(* CODESYS project BasePpt.library
   Company: Vistaprint
   Version: 0.0.0.76
   Description: 0.0.0.76	- IBH simulation improvements
      0.0.0.75	- new BaseConcept and BaseElements
      	- add full simulation to IBH
      	- remove simulation from OVN
      	- JCL clears Cleaning request in OFFbusy and MaintenanceMode
      0.0.0.74	- new BaseConcept and BaseElements
      0.0.0.73	- new BaseConcept and BaseElements
      0.0.0.72	- new BaseElements
      0.0.0.71	- JCL fix, Oven tracking band2 must be off for 3 cycles
      0.0.0.70	- PBC: Different SheetToSheet times for Auto & Manual Mode
      	- JCL: Rework Manual behavior
      0.0.0.69	- JCL: Take the message buffer out of the CUR
      0.0.0.68	- JCL: Error Exit Error fixed
      0.0.0.67	- JCL: Fix for Manual Mode Exit
      0.0.0.66	- JCL: added EOFF, changed PON
      0.0.0.65	- Added new BaseElements
      	- better DeStacker error msg
      0.0.0.64	- Added new BaseElements
      	- Added Manual State to JCL
      	- Adapted UMC usage in all controllers
      0.0.0.63	- GRR only showing 1 error when connection lost
      0.0.0.62	- PBC: changed buffer counter to int
      0.0.0.61	- DeStacker checks if empty
      0.0.0.60	- when DoubleSheet only Warning when turned off on DeStacker
      0.0.0.59	- BCH can go back to RUN from ERROR
      0.0.0.58	- BCH + JCL fixes
      0.0.0.57	- option to not wait for paper in OVN.OFFBusy
      	- support AnalogValue on GRR
      0.0.0.56	- fixed OVN.OFFBusy time calculation
      0.0.0.55	- JCL check Jetter state in RUN
      	- latest BaseConcept and BaseElements
      	- OVN wait in OFFBusy until sheets are out
      0.0.0.54	- TCP - Fix for constant resend of command
      0.0.0.53	- fixes
      0.0.0.52	- TCP - Introduced automatic reconnect
      0.0.0.51	- PBC - Fix for StopDestacking and Manual mode.
      0.0.0.50	- OVN has TSTOP when settings change
      0.0.0.49	- Saber PBC StopBit modification, different PBC alarm handling
      0.0.0.48	- small fixes for DeStacker
      0.0.0.47	- GRR warning automatically disappear
      0.0.0.46	- TCP.CtrlInit-Added call to super
      0.0.0.45	- manual operation on GRR is only a WARNING
      0.0.0.44	- OVN recovers from EOFF by reconnecting IBHLink
      0.0.0.43	- ignore bolStopReleaseItems when in manual mode
      0.0.0.42	- namechange GRN to GRR, ToggleBit for GRR
      0.0.0.41   - StopReleaseItems for PBC
      0.0.0.40	- new BaseElements
      0.0.0.39	- added CtrlSIf and strFullName where missing, new libraries
      0.0.0.38	- Better GRN error msgs
      0.0.0.37	- PBC Fixes
      0.0.0.36	- PTS Error Message Fixed
      	- PBC EvaluateEject fix
      	- PST Eject paper if not finished
      0.0.0.35	- Add long term test to PTS
      0.0.0.34 	- Pts fix when using with Servo
      0.0.0.33 	- Upgraded to newest TC 3.1 4016.12
      	- Upgraded all Libraries
      0.0.0.32 - Bug fixes in PTS and POD
      0.0.0.31 - BaseElements V0.0.1.30 referred
      0.0.0.30 - updated Oven and IBH
      0.0.0.29 - Fix PTS warning bug
      0.0.0.28 - Added a new version of the PBC
      0.0.0.27 - added strFullName
      0.0.0.26 - Added RAX, POD, TCP, PST, Updated PBC, PTS
      0.0.0.25 - Added the newest Base + Elements + TC 3.1 4016.6
      0.0.0.24 - Added the newest Base + Elements
      0.0.0.23 - Updated to TwinCat 4016.5
      0.0.0.22 - FB_PTB Always SingleAnswer
      0.0.0.21 - Added newest Elemets Library 
      0.0.0.20 - Added newest Elemets Library and reworked CtrlInit
      0.0.0.19 - Added newest Elemets Library
      0.0.0.18 - Added newest revision of the PTS
      
      0.0.0.16 - Added new Base and Elements 
      0.0.0.15 - Added new Base and Elements 
      0.0.0.14 - Added new Base and Elements 
      0.0.0.13 - Added new Base and Elements 
      0.0.0.11 - Added new Base and Elements library
      0.0.0.10 - PCE: no EOFF State!! in EOFF go to OFF (in Always); Redo changes of 0.0.0.6; PTS.Always no EOFF; sta_OFFBusy in PTS reworked;
      0.0.0.9 - Merged the DeStacker MDC with the BasePpt MDC
      0.0.0.8 - Added newer Versions of libraries.
      0.0.0.7 - Added newer Versions of libraries.
      0.0.0.6 - Changes for Simualtion in MDC, sta_OFFBusy in PTB/MDC reworked; Always in PTB reworked;
      0.0.0.5 - Added new Base_PLC 0.3.4.1
      0.0.0.4 - Bug fixed in FB_PTB
      0.0.0.3 - Update to take the newest libraries 
      0.0.0.2 - Update to Base_PLC 0.3.3.2; Update to Base_Elements 0.0.0.9
   Author: pcipriano
   Title: BasePpt

Project tree, tasks and I/O mapping:
  libraries: Base_Elements, 0.0.1.50 (Vistaprint); Base_PLC, 0.3.5.12 (Vistaprint); Tc2_EtherCAT, 3.3.3.0 (Beckhoff Automation GmbH); Tc2_MC2, 3.3.8.0 (Beckhoff Automation GmbH); Tc2_S5S7Com, 3.3.0.0 (Beckhoff Automation GmbH); Tc2_Standard, 3.3.0.0 (Beckhoff Automation GmbH); Tc2_System, 3.3.8.1 (Beckhoff Automation GmbH); Tc2_TcpIp, 3.3.2.0 (Beckhoff Automation GmbH); Tc2_Utilities, 3.3.8.0 (Beckhoff Automation GmbH); Tc3_Interfaces, 3.3.0.0 (Beckhoff Automation GmbH); Tc3_MemMan, 3.3.1.0 (Beckhoff Automation GmbH); Tc3_Module, 3.3.6.0 (Beckhoff Automation GmbH)
  GVLs/
    global variables Constants
  POUs/
    Controller/
      Driver/
        IBH (IBH Link)/
          function block FB_IBH [ST]: Always, bitAccess, CtrlInit, CtrlSIf, FB_init, getCmdState, getCtrlSIf, setAckError, setAirflow, setBeltOn, setOff, setRun, setSpeed, setStandby, setTemp, sta_CONNECT, sta_CONNECTBusy, sta_DISCONNECT, sta_DISCONNECTBusy, sta_OFF, sta_OFFBusy, sta_PON, sta_PONBusy, sta_READ, sta_READBusy, sta_WRITE, sta_WRITEBusy, StateMachine
          global variables IBH_CmdState
          data type T_Ctrl_SIf_IBH
          data type T_Ctrl_SIf_IBH_Cfg
          data type T_Ctrl_SIf_IBH_Cur
          data type T_Ctrl_SIf_IBH_Par
        POD (PLCopen Driver)/
          data type E_AmpType
          data type E_POD_UseHomeSwitch
          data type E_ValueType
          function block FB_POD [ST]: AD_SIf, CtrlInit, CycleEndDuty, CycleStartDuty, getCmdState, sJobReadParameter, sJobReadParameterNC, sJobWriteParameter, sJobWriteParameterNC, sta_AbsMoveBusy, sta_Error, sta_HomeBusy, sta_ModMoveBusy, sta_NegJogBusy, sta_NegMoveBusy, sta_PosJogBusy, sta_PosMoveBusy, sta_PowerOff, sta_PowerOnBusy, sta_QStopBusy, sta_RelMoveBusy, sta_StopBusy, sta_WaitForJob, StateMachine, StateMachine_Service
          global variables POD_Cmd
          global variables POD_Const
          data type T_POD
          data type T_POD_Cfg
          data type T_POD_DigitalInputs
          data type T_POD_Error
          data type T_POD_Move
          data type T_POD_Service
          data type T_POD_StateMachine
          data type T_POD_Status
          data type T_POD_StatusWord
        PTR [Paper Tracker]/
          data type E_PTR_Status
          function block FB_PTR [ST]: BeltLength, EnterComplete, FB_init, Insert, PaperEntryOffset, PaperOnBelt, Pop, PositionList, Push, Reset, TimeBase
          data type T_PTR_STRUCT
        TCP (TCP communication driver)/
          data type E_ALM_TCP
          function block FB_TCP [ST]: Always, CtrlInit, CtrlSIf, CycleEndDuty, CycleStartDuty, FB_init, getCmdState, getCtrlSIf, M_Pop, M_Push, ReceiveDataSequence, SendDataSequence, sta_CLOSE, sta_CLOSEBusy, sta_CONNECT, sta_CONNECTBusy, sta_ERROR, sta_ERRORQuit, StateMachine
          data type ST_Header
          data type T_Ctrl_SIf_TCP
          data type T_Ctrl_SIf_TCP_Cfg
          data type T_Ctrl_SIf_TCP_Cur
          data type T_Ctrl_SIf_TCP_Par
          global variables TCP_CmdState
          global variables TCP_Constants
      Lvl0/
        GRR (Granulate Remote)/
          helper/
            function cycle_Grr [ST]
            function init_Grr [ST]
            data type T_GRR
            data type T_GRR_CTRL
            data type T_GRR_ID
            data type T_GRR_IO
          data type E_ALM_GRR
          function block FB_GRR [ST]: Always, CtrlSIf, FB_init, getCtrlSIf, IoInBridge, IoOutBridge, sta_ERROR, sta_ERRORQuit, sta_OFF, sta_OFFBusy, sta_PON, sta_PONBusy, sta_RUN, sta_RUNBusy, StateMachine
          data type T_Ctrl_SIf_GRR
          data type T_Ctrl_SIf_GRR_Cfg
          data type T_Ctrl_SIf_GRR_Cur
          data type T_Ctrl_SIf_GRR_In
          data type T_Ctrl_SIf_GRR_Out
          data type T_Ctrl_SIf_GRR_Par
        JCL (Jetter Client)/
          helper/
            function cycle_Jcl [ST]
            function init_Jcl [ST]
            data type T_JCL
            data type T_JCL_CTRL
            data type T_JCL_ID
            data type T_JCL_IO
          data type E_ALM_JCL
          function block FB_JCL [ST]: Always, checkChildAlmClass, cmdCALIBRATION, cmdCLEAN, cmdOFF, cmdPON, cmdRUN, cmdSTANDBY, CtrlInit, CtrlSIf, FB_init, getCmdState, getCtrlSIf, HandleReceiveData, RequestState, ResetAlarms, sta_CALIBRATION, sta_CALIBRATIONBusy, sta_CLEANING, sta_CLEANINGBusy, sta_CONNECTBusy, sta_EOFF, sta_EOFFBusy, sta_ERROR, sta_ERRORQuit, sta_MANUALMODE, sta_OFF, sta_OFFBusy, sta_PON, sta_PONBusy, sta_RUN, sta_RUNBusy, sta_STANDBY, sta_STANDBYBusy, StateMachine, TCP
          global variables JCL_CmdState
          global variables JCL_Constants
          data type T_Ctrl_SIf_JCL
          data type T_Ctrl_SIf_JCL_Cfg
          data type T_Ctrl_SIf_JCL_Cur
          data type T_Ctrl_SIf_JCL_Par
          data type T_JCL_AlmMsg
          data type T_JCL_Command
          data type T_JCL_PrintDone
          data type T_JCL_RequestCleaning
          data type T_JCL_State
          data type U_JCL_Message
        RAX(Rotative Axis)/
          data type E_ALM_RAX
          function block FB_RAX [ST]: Always, CtrlSIf, FB_init, getCmdState, getDirection, IoOutBridge, sta_EOFF, sta_EOFFBusy, sta_ERROR, sta_ERRORQuit, sta_INIT, sta_INITBusy, sta_JOG_NEG, sta_JOG_POS, sta_OFF, sta_OFFBusy, sta_POS, sta_POSBusy, sta_REL_POS, sta_REL_POSBusy, sta_STOP, sta_STOPBusy, sta_Turn, sta_TurnBusy, StateMachine
          function fSetPar [ST]
          global variables RAX_CmdState
          data type T_Ctrl_SIf_RAX
          data type T_Ctrl_SIf_RAX_Cfg
          data type T_Ctrl_SIf_RAX_Cur
          data type T_Ctrl_SIf_RAX_Ilk
          data type T_Ctrl_SIf_RAX_Par
      Lvl1/
        BCH (Barcode with DataChannel)/
          helper/
            function cycle_Bch [ST]
            function init_Bch [ST]
            data type T_BCH
            data type T_BCH_CTRL
            data type T_BCH_DATACHN
            data type T_BCH_ID
            data type T_BCH_IO
          global variables BCH_CmdState
          data type E_ALM_BCH
          function block FB_BCH [ST]: Always, BarcodeReader, CtrlInit, CtrlSIf, DataChannel, FB_init, getCmdState, getCtrlSIf, IoInBridge, sta_ERROR, sta_ERRORQuit, sta_OFF, sta_OFFBusy, sta_RUN, sta_RUNBusy, StateMachine
          data type T_Ctrl_SIf_BCH
          data type T_Ctrl_SIf_BCH_Cfg
          data type T_Ctrl_SIf_BCH_Cur
          data type T_Ctrl_SIf_BCH_In
          data type T_Ctrl_SIf_BCH_Par
        MDC [Malteser Drive Controller]/
          data type E_ALM_MDC
          function block FB_MDC [ST]: ActualPosition, Always, CtrlInit, CtrlSIf, Drive, FB_init, getCmdState, getCtrlSIf, GetTurningDirection, IncrementPosition, IoInBridge, IoOutBridge, SetPositionToGo, sta_ERROR, sta_ERRORQuit, sta_InitializeBusy, sta_InPosition, sta_InPositionBusy, sta_OFF, sta_OFFBusy, sta_PON, sta_PREPOSITION, sta_PREPOSITIONbusy, sta_StartTurnBusy, sta_TurnBusy, sta_TURNDONE, StateMachine
          global variables MDC_CmdState
          data type T_Ctrl_SIf_MDC
          data type T_Ctrl_SIf_MDC_Cfg
          data type T_Ctrl_SIf_MDC_Cur
          data type T_Ctrl_SIf_MDC_Ilk
          data type T_Ctrl_SIf_MDC_In
          data type T_Ctrl_SIf_MDC_Out
          data type T_Ctrl_SIf_MDC_Par
        OVN (Oven)/
          helper/
            function cycle_Ovn [ST]
            function init_Ovn [ST]
            data type T_OVN
            data type T_OVN_CTRL
            data type T_OVN_DATACHN
            data type T_OVN_ID
            data type T_OVN_IO
          data type E_ALM_OVN
          function block FB_MONITOR [ST]: resetTime
          function block FB_OVN [ST]: Always, checkParameter, chooseTesomaErrors, CtrlInit, CtrlSIf, DataChannel, FB_init, getCmdState, getCtrlSIf, IBH, sta_BELTONLY, sta_BELTONLYBusy, sta_ERROR, sta_ERRORQuit, sta_OFF, sta_OFFBusy, sta_PON, sta_PONBusy, sta_RUN, sta_RUNBusy, StateMachine
          function block FB_Tracker [ST]: addElement, DataChannel, deleteAll, deleteElement, distanceAfterOven_mm, distanceBeforeOven_mm, markAllTrash, moduleLength_mm, numberOfElements, numberOfModules, sampleTime_us, sendData, update
          global variables OVN_CmdState
          data type T_Ctrl_SIf_OVN
          data type T_Ctrl_SIf_OVN_Cfg
          data type T_Ctrl_SIf_OVN_Cur
          data type T_Ctrl_SIf_OVN_In
          data type T_Ctrl_SIf_OVN_Out
          data type T_Ctrl_SIf_OVN_Par
          data type T_Data
        PTA [Paper Transport Alignment]/
          helper/
            function cycle_Pta [ST]
            function init_Pta [ST]
            data type T_PTA
            data type T_PTA_CTRL
            data type T_PTA_ID
            data type T_PTA_IO
        PTB [Paper Transport Belt]/
          BeltParameterFunction/
            data type T_Belt_Cfg_Base
            data type T_Belt_Cur_Base
            data type T_Belt_Par_Base
          helper/
            function cycle_Ptb [ST]
            function init_Ptb [ST]
            data type T_PTB
            data type T_PTB_CTRL
            data type T_PTB_ID
            data type T_PTB_IO
          data type E_ALM_PTB
          data type E_BELT_DIRECTION
          data type E_PTB_MODE
          data type E_PTB_PaperDirection
          function block FB_PTB [ST]: Always, CalculateBeltParameter, CalculateModeParameter, CheckPumpState, cmd_OFF, cmd_RUN, cmd_STOP, CtrlInit, CtrlSIf, Drive, FB_init, getCmdState, getCtrlSIf, IoInBridge, IoOutBridge, PaperPositionHandling, PositionList, SetPumpComand, sta_EJECTPAPER, sta_EJECTPAPERbusy, sta_ERROR, sta_ERRORQuit, sta_OFF, sta_OFFBusy, sta_PON, sta_RUN, sta_RUNBusy, sta_STACKPAPER, sta_STACKPAPERbusy, sta_STOP, sta_STOPBusy, StateMachine, VacuumPump
          global variables PTB_CmdState
          data type T_Ctrl_SIf_PTB
          data type T_Ctrl_SIf_PTB_Cfg
          data type T_Ctrl_SIf_PTB_Cur
          data type T_Ctrl_SIf_PTB_Ilk
          data type T_Ctrl_SIf_PTB_In
          data type T_Ctrl_SIf_PTB_Out
          data type T_Ctrl_SIf_PTB_Par
      Lvl2/
        PBC [Paper Buffer Controller]/
          helper/
            function cycle_Pbc [ST]
            function init_Pbc [ST]
            data type T_PBC
            data type T_PBC_CTRL
            data type T_PBC_ID
            data type T_PBC_IO
          data type E_ALM_PBC
          function block FB_PBC [ST]: Always, Belt, CountPaper, CtrlInit, CtrlSIf, DeStacker, FB_init, getCmdState, getCtrlSIf, IoInBridge, IoOutBridge, PaperHight, PaperWidth, sta_ERROR, sta_ERRORQuit, sta_INITbusy, sta_OFF, sta_OFFBusy, sta_PON, sta_RUN, sta_RUNbusy, sta_STOP, sta_STOPbusy, StateMachine
          global variables PBC_CmdState
          data type T_Ctrl_SIf_PBC
          data type T_Ctrl_SIf_PBC_Cfg
          data type T_Ctrl_SIf_PBC_Cur
          data type T_Ctrl_SIf_PBC_Ilk
          data type T_Ctrl_SIf_PBC_In
          data type T_Ctrl_SIf_PBC_Out
          data type T_Ctrl_SIf_PBC_Par
        PCE [Paper Belt Corner Element]/
          helper/
            function cycle_Pce [ST]
            function init_Pce [ST]
            data type T_PCE
            data type T_PCE_CTRL
            data type T_PCE_ID
            data type T_PCE_IO
          data type E_ALM_PCE
          function block FB_PCE [ST]: Always, CtrlInit, CtrlSIf, DriveIn, DriveOut, FB_init, getCmdState, getCtrlSIf, IoInBridge, IoOutBridge, PaperExitValveActive, PaperInputValveActive, sta_ERROR, sta_ERRORQuit, sta_OFF, sta_OFFBusy, sta_PON, sta_RUN, sta_RUNBusy, sta_STOP, sta_STOPBusy, StateMachine
          global variables PCE_CmdState
          data type T_Ctrl_SIf_PCE
          data type T_Ctrl_SIf_PCE_Cfg
          data type T_Ctrl_SIf_PCE_Cur
          data type T_Ctrl_SIf_PCE_Ilk
          data type T_Ctrl_SIf_PCE_In
          data type T_Ctrl_SIf_PCE_Out
          data type T_Ctrl_SIf_PCE_Par
        PST [Paper Stacker]/
          helper/
            function cycle_Pst [ST]
            function init_Pst [ST]
            data type T_PST
            data type T_PST_CTRL
            data type T_PST_ID
            data type T_PST_IO
          data type E_ALM_PST
          function block FB_PST [ST]: Always, Belt, CtrlInit, CtrlSIf, FB_init, getCmdState, getCtrlSIf, IoInBridge, PaperStackSendFifo, sta_EJECTBusy, sta_OFF, sta_OFFBusy, sta_RUN, sta_RUNBusy, StateMachine
          global variables PST_CmdState
          data type T_Ctrl_SIf_PST
          data type T_Ctrl_SIf_PST_Cfg
          data type T_Ctrl_SIf_PST_Cur
          data type T_Ctrl_SIf_PST_In
          data type T_Ctrl_SIf_PST_Par
          data type T_ItemPaperInfo
        PTS [Paper Turning Station]/
          helper/
            function cycle_Pts [ST]
            function init_Pts [ST]
            data type T_PTS
            data type T_PTS_CTRL
            data type T_PTS_ID
            data type T_PTS_IO
          data type E_ALM_PTS
          data type E_PTS_MODE
          function block FB_PTS [ST]: Always, Belt, CalculateOutputDelay, ChangeDistributionModeParameter, CtrlInit, CtrlSIf, FB_init, getCmdState, getCtrlSIf, GetItemBusy, IoInBridge, IoOutBridge, Malteser, Servo, sta_ERROR, sta_ERRORQuit, sta_GetItemBusy, sta_InitializeBusy, sta_OFF, sta_OFFBusy, sta_PaperDelayBusy, sta_PON, sta_RUN, sta_RUNBusy, sta_STANDBY, sta_STANDBYBusy, sta_STOP, sta_STOPbusy, sta_TurnEmptyBusy, sta_TurnPaperBusy, sta_WaitPaper, sta_WaitPaperGone, StateMachine
          global variables PTS_CmdState
          global variables PTS_Persistent
          data type T_Ctrl_SIf_PTS
          data type T_Ctrl_SIf_PTS_Cfg
          data type T_Ctrl_SIf_PTS_Cur
          data type T_Ctrl_SIf_PTS_Ilk
          data type T_Ctrl_SIf_PTS_In
          data type T_Ctrl_SIf_PTS_Out
          data type T_Ctrl_SIf_PTS_Par
          data type T_PTS_InOutPositions
      Lvl3/
      Lvl4/
      Top/
      Utility/
        Data Channel/
          OvenMessage/
            function block FB_OvenSendDch [ST]: InitChannel, SendData
            global variables OvenConst
            data type T_Oven_DCH
            data type T_OvenSendData
        FiFo/
          function block FB_DataSetFifo [ST]: A_Add, A_Get, A_Remove, A_Reset
        LookupTable/
          function block FB_LookupTable [ST]: A_Add, A_LookupByKey, A_LookupByValue, A_RemoveKey, A_Reset
          global variables LUT_Constants
  Version/
    global variables Global_Version
*)

// POUs/Controller/Driver/IBH (IBH Link)/T_Ctrl_SIf_IBH
TYPE T_Ctrl_SIf_IBH :
STRUCT
	///configuration
	Cfg: T_Ctrl_SIf_IBH_Cfg;
	///parameter
	Par: T_Ctrl_SIf_IBH_Par;
	///current values
	Cur: T_Ctrl_SIf_IBH_Cur;
END_STRUCT
END_TYPE

// POUs/Controller/Driver/IBH (IBH Link)/T_Ctrl_SIf_IBH_Cfg
TYPE T_Ctrl_SIf_IBH_Cfg :
STRUCT
	/// Number of Modules in use, <= 8 
	uiNumberOfModules: UINT;
	/// IPv4 network address 
	tIpAddress: T_IPv4Addr;
	/// Remote (server) port address 
	udiPortAdress: UDINT;
	/// MPI device address 
	nDeviceAddress: BYTE;
	/// Read/write from/to datablock number 
	nDatablockNumber: BYTE;
	/// Maximum time allowed for the execution of the command 
	tTimeout: TIME;
	/// Write byte/word offset/start address 
	nWriteStartAddress: WORD;
	/// Read byte/word offset/start address 
	nReadStartAddress: WORD;
	uiByteOffset_rd_iStatus: UINT;
	uiByteOffset_rd_bOff: UINT;
	uiBitOffset_rd_bOff: UINT;
	uiByteOffset_rd_bBeltOn: UINT;
	uiBitOffset_rd_bBeltOn: UINT;
	uiByteOffset_rd_bManual: UINT;
	uiBitOffset_rd_bManual: UINT;
	uiByteOffset_rd_bRun: UINT;
	uiBitOffset_rd_bRun: UINT;
	uiByteOffset_rd_bSetParam: UINT;
	uiBitOffset_rd_bSetParam: UINT;
	uiByteOffset_rd_bGetParam: UINT;
	uiBitOffset_rd_bGetParam: UINT;
	uiByteOffset_rd_bAckError: UINT;
	uiBitOffset_rd_bAckError: UINT;
	uiByteOffset_rd_adiTemp_mc: UINT;
	uiByteOffset_rd_adiAir_p: UINT;
	uiByteOffset_rd_diSpeed_mm_min: UINT;
	uiByteOffset_rd_iErrorLevel: UINT;
	uiByteOffset_rd_iErrorID: UINT;
	uiByteOffset_rd_iErrorValue: UINT;
	uiByteOffset_wr_iOff: UINT;
	uiByteOffset_wr_iBeltOn: UINT;
	uiByteOffset_wr_iManual: UINT;
	uiByteOffset_wr_iRun: UINT;
	uiByteOffset_wr_iSetParam: UINT;
	uiByteOffset_wr_iGetParam: UINT;
	uiByteOffset_wr_iAckError: UINT;
	uiByteOffset_wr_adiTemp_mc: UINT;
	uiByteOffset_wr_adiAir_p: UINT;
	uiByteOffset_wr_diSpeed_mm_min: UINT;
END_STRUCT
END_TYPE

// POUs/Controller/Driver/IBH (IBH Link)/T_Ctrl_SIf_IBH_Cur
TYPE T_Ctrl_SIf_IBH_Cur :
STRUCT
END_STRUCT
END_TYPE

// POUs/Controller/Driver/IBH (IBH Link)/T_Ctrl_SIf_IBH_Par
TYPE T_Ctrl_SIf_IBH_Par :
STRUCT
END_STRUCT
END_TYPE

// POUs/Controller/Driver/POD (PLCopen Driver)/E_AmpType
TYPE E_AmpType :
(
	BOTH_ROT_LIN := 0,
	ROTARY_AMP := 1,
	LINEAR_AMP := 2
) USINT;
END_TYPE

// POUs/Controller/Driver/POD (PLCopen Driver)/E_POD_UseHomeSwitch
TYPE E_POD_UseHomeSwitch :
(
	FUB_Input := 0,
	HomeSwitch,
	/// internal IO 2 Home switch 					0: Switched off, 1: Switched on
	SI0,
	/// internal IO 16 SI0:				0: Switched off (Open),1: Switched on (Close)
	SI1,
	/// internal IO 17 SI0:				0: Switched off (Open),1: Switched on (Close)
	SI2,
	/// internal IO 18 SI0:			0: Switched off (Open),1: Switched on (Close)
	SI3,
	/// internal IO 19 SI0:				0: Switched off (Open),1: Switched on (Close)
	SI4,
	/// internal IO 20 SI0:					0: Switched off (Open),1: Switched on (Close)
	SI5,
	/// internal IO 21 SI0:	 				0: Switched off (Open),1: Switched on (Close)
	/// internal IO 22 SI0:					0: Switched off (Open),1: Switched on (Close)
	SI6
) USINT;
END_TYPE

// POUs/Controller/Driver/POD (PLCopen Driver)/E_ValueType
TYPE E_ValueType :
(
	TYPE_NOT_SPECIFIED := 0,
	TYPE_SINT := 1,
	TYPE_INT := 2,
	TYPE_DINT := 3,
	TYPE_USINT := 4,
	TYPE_UINT := 5,
	TYPE_UDINT := 6,
	TYPE_STRING := 7
) USINT;
END_TYPE

// POUs/Controller/Driver/POD (PLCopen Driver)/T_POD
TYPE T_POD :
STRUCT
	strAxisName: STRING(31);
	strState: STRING;
	strCmd: STRING;
	intCmd: INT;
	intServiceCmd: INT;
	stStatus: T_POD_Status;
	stMove: T_POD_Move;
	stErr: T_POD_Error;
	stCfg: T_POD_Cfg;
	stService: T_POD_Service;
END_STRUCT
END_TYPE

// POUs/Controller/Driver/POD (PLCopen Driver)/T_POD_Cfg
TYPE T_POD_Cfg :
STRUCT
	bolSimulation: BOOL;
	///>0 Homeposition set if calibsignal active
	lreHomePosition: LREAL;
	/// Home Mode
	eHomingMode: MC_HomingMode;
	/// define home switch: 0 use FUB input, 
	eUseHomeSwitch: E_POD_UseHomeSwitch;
END_STRUCT
END_TYPE

// POUs/Controller/Driver/POD (PLCopen Driver)/T_POD_DigitalInputs
TYPE T_POD_DigitalInputs :
STRUCT
	///0 N-OT: 	Negative limit switch 	0: Switched off, 1: Switched on
	bol_N_OT: BOOL;
	///1 P-OT: 	Positive limit switch 	0: Switched off, 1: Switched on
	bol_P_OT: BOOL;
	///2 Home switch 					0: Switched off, 1: Switched on
	bol_HomeSwitch: BOOL;
	///16 SI0:	CN1-13pin 				0: Switched off (Open),1: Switched on (Close)
	bol_SI0: BOOL;
	///17 SI1:	CN1-7pin 				0: Switched off (Open),1: Switched on (Close)
	bol_SI1: BOOL;
	///18 SI2:	CN1-8pin 				0: Switched off (Open),1: Switched on (Close)
	bol_SI2: BOOL;
	///19 SI3:	CN1-9pin 				0: Switched off (Open),1: Switched on (Close)
	bol_SI3: BOOL;
	///20 SI4:	CN1-10pin 				0: Switched off (Open),1: Switched on (Close)
	bol_SI4: BOOL;
	///21 SI5:	CN1-11pin 				0: Switched off (Open),1: Switched on (Close)
	bol_SI5: BOOL;
	///22 SI6:	CN1-12pin 				0: Switched off (Open),1: Switched on (Close)
	bol_SI6: BOOL;
END_STRUCT
END_TYPE

// POUs/Controller/Driver/POD (PLCopen Driver)/T_POD_Error
TYPE T_POD_Error :
STRUCT
	/// Reset failure
	bolErrAck: BOOL;
	/// atleast one failure active
	bolErrorActive: BOOL;
	/// error in MC fub error
	bolMCError: BOOL;
	/// error in NC (motion controller)
	bolNCError: BOOL;
	/// error in drive (ELMO)
	bolDriveError: BOOL;
	/// error ID
	dwoErrorID: DWORD;
END_STRUCT
END_TYPE

// POUs/Controller/Driver/POD (PLCopen Driver)/T_POD_Move
TYPE T_POD_Move :
STRUCT
	///target position [Units] 
	lreSetPos: LREAL;
	/// Direction used for Modulo position
	eDirection: MC_Direction;
	///set speed [Units/s] 
	lreSetSpeed: LREAL;
	///set acc  [Units/s^2] 
	lreSetAcc: LREAL;
	///set dec  [Units/s^2] 
	lreSetDec: LREAL;
	///set dec  [Units/s^2] quickstop
	lreSetDecFast: LREAL;
	///lreSetDec : DINT; //set dec  [Units/s^2] 
	lreSetJerk: LREAL;
	/// speed override for all drive commands (0 ≤Override≤ 100.0)
	lreSpeedOverride: LREAL := 100.0;
	lreSWLimitNeg_mm: LREAL;
	lreSWLimitPos_mm: LREAL;
	/// Actual position [Units] 
	lreActPos: LREAL;
	/// Actual modulo position [Units] 
	lreActModPos: LREAL;
	/// act speed [Units/s] 
	lreActVel: LREAL;
	/// [Nm] actual torque The torque actual value corresponds to the instantaneous torque in the drive motor. The value is given in units of per thousand of rated torque.
	lreActTorque: LREAL;
END_STRUCT
END_TYPE

// POUs/Controller/Driver/POD (PLCopen Driver)/T_POD_Service
TYPE T_POD_Service :
STRUCT
	/// Index of the object that should be written to.
	worIndex: WORD;
	/// Sub-index of the object that should be written to.
	bytSubIndex: BYTE;
	/// Address (pointer) of the send buffer.
	dwo_pSrcBuf: DWORD;
	/// Number (in bytes) of data to be sent.
	udi_cbBufLen: UDINT;
	/// value type
	eValueType: E_ValueType;
	/// parameter number of read/write NC parameters
	eNC_ParNumber: MC_AxisParameter;
	/// write/read value if dwo_pSrcBuf = 0
	strValue: STRING;
END_STRUCT
END_TYPE

// POUs/Controller/Driver/POD (PLCopen Driver)/T_POD_StateMachine
TYPE T_POD_StateMachine :
STRUCT
	///actual state
	intState: INT;
	///state of last cycle
	intStateLastCycle: INT;
	///save history backup p.e. in ERROR state
	intStateHistory: INT;
	///set state for next cycle
	intStateNext: INT;
END_STRUCT
END_TYPE

// POUs/Controller/Driver/POD (PLCopen Driver)/T_POD_Status
TYPE T_POD_Status :
STRUCT
	/// Hardware enable:0 = Open 1 = Closed  
	bolEnable: BOOL;
	/// 1 = Network initialized  
	bolNetwOk: BOOL;
	/// 1 = Initialization done 
	bolInitOk: BOOL;
	bolReady: BOOL;
	/// 1 = Controller switched on  
	bolCtrlOn: BOOL;
	/// 1 = Homing done  
	bolHomeOk: BOOL;
	/// 1 = In position (target position reached)  
	bolInPos: BOOL;
	/// 1 = Axis moving  
	bolMoving: BOOL;
	/// 1 = negativ endswitch active -> no movement negative allowed
	bolNegHWSwitch: BOOL;
	/// 1 = positive endswitch active -> no movement positive allowed
	bolPosHWSwitch: BOOL;
	/// 1 = negativ endswitch active -> no movement negative allowed
	bolNegSWSwitch: BOOL;
	/// 1 = positive endswitch active -> no movement positive allowed
	bolPosSWSwitch: BOOL;
	/// drive digital inputs of elmo drive
	stDigIn: T_POD_DigitalInputs;
END_STRUCT
END_TYPE

// POUs/Controller/Driver/POD (PLCopen Driver)/T_POD_StatusWord
TYPE T_POD_StatusWord :
STRUCT
	/// 0	Ready TO Switch on =1
	bolReadyToSwitchOn: BOOL;
	///1	Switched on =1
	bolSwitchedOn: BOOL;
	///2	Operation enabeld =1
	bolOperationEnabled: BOOL;
	///3	Fault/Fault Reaction
	bolFault: BOOL;
	///4	MainPower on =1
	bolMainPowerOn: BOOL;
	///5	Quickstop inaktive =1
	bolQuickStopInactive: BOOL;
	///6	Switch on disabled =1
	bolSwitchOnDisabled: BOOL;
	///7	Warning is occurred =1
	bolWarning: BOOL;
	///8	not used always 0
	bolBit08: BOOL;
	///9	The Remote bit is always set by the Elmo servo drive
	bolRemote: BOOL;
	///10	Target Reached
	bolTargetReached: BOOL;
	///11	Internal Limit active =1
	bolInternLimit: BOOL;
END_STRUCT
END_TYPE

// POUs/Controller/Driver/PTR [Paper Tracker]/E_PTR_Status
TYPE E_PTR_Status :
(
	EnterBusy,
	OnBelt,
	ExitBusy,
	Gone,
	ERROR,
	MAX_E_PTR_Status
);
END_TYPE

// POUs/Controller/Driver/PTR [Paper Tracker]/T_PTR_STRUCT
TYPE T_PTR_STRUCT :
STRUCT
	// [us] Time of the paper on the belt
	udiTimeOnBelt_us				: UDINT;
	// [mm] Position of the paper on the belt
	lrePositionOnBelt_mm			: LREAL;
	// [mm] Position of the paper on the belt Adjusted to the possible maximum
	lrePositionOnBeltAdjusted_mm	: LREAL;
	// Paper Item Id
	udiItemId						: UDINT;
	// Error	
	eStatus							: E_PTR_Status;
END_STRUCT
END_TYPE

// POUs/Controller/Driver/TCP (TCP communication driver)/E_ALM_TCP
TYPE E_ALM_TCP :
(
	SocketConnectionLost := 1,
	AddToSendBufferFailed := 2,
	RemoveFromSendBufferFailed := 3,
	GetFromSendBufferFailed := 4,
	AddToReceiveBufferFailed := 5,
	RemoveFromReceiveBufferFailed := 6,
	GetFromReceiveBufferFailed := 7,
	NotSent := 8,
	NoAckReceived := 9,
	FubErrorClientConnection := 10,
	FubErrorSendData := 11,
	FubErrorReceiveData := 12,
	MAX_E_ALM_TCP
) UINT;
END_TYPE

// POUs/Controller/Driver/TCP (TCP communication driver)/ST_Header
{attribute 'pack_mode' := '1'}
TYPE ST_Header :
STRUCT
	uinMsgId: UINT;
	udiMsgSize: UDINT;
END_STRUCT
END_TYPE

// POUs/Controller/Driver/TCP (TCP communication driver)/T_Ctrl_SIf_TCP
TYPE T_Ctrl_SIf_TCP :
STRUCT
	/// configuration
	Cfg: T_Ctrl_SIf_TCP_Cfg;
	/// parameter
	Par: T_Ctrl_SIf_TCP_Par;
	/// current values
	Cur: T_Ctrl_SIf_TCP_Cur;
	/// alarm number used in this controller
	Alm: ARRAY[1..(E_ALM_TCP.MAX_E_ALM_TCP - 1)] OF T_Ctrl_Alm;
END_STRUCT
END_TYPE

// POUs/Controller/Driver/TCP (TCP communication driver)/T_Ctrl_SIf_TCP_Cfg
TYPE T_Ctrl_SIf_TCP_Cfg :
STRUCT
	/// depending on the protocol an ACK is used or not
	bUsingAck: BOOL;
	/// Enable Auto Reconnect
	bolAutoReconnectEnable: BOOL;
END_STRUCT
END_TYPE

// POUs/Controller/Driver/TCP (TCP communication driver)/T_Ctrl_SIf_TCP_Cur
TYPE T_Ctrl_SIf_TCP_Cur :
STRUCT
	bolFubErrorActive: BOOL;
END_STRUCT
END_TYPE

// POUs/Controller/Driver/TCP (TCP communication driver)/T_Ctrl_SIf_TCP_Par
TYPE T_Ctrl_SIf_TCP_Par :
STRUCT
	strIPAdr: STRING(15);
	udiPort: UDINT;
	tTOConnection: TIME;
	tTOReceive: TIME;
	tTOSend: TIME;
	iMaxWaitTimeAck: TIME;
	iMaxSendTry: USINT;
END_STRUCT
END_TYPE

// POUs/Controller/Lvl0/GRR (Granulate Remote)/helper/T_GRR
TYPE T_GRR :
STRUCT
	io:		T_GRR_IO;
	ctrl:	T_GRR_CTRL;
	id:		T_GRR_ID;
END_STRUCT
END_TYPE

// POUs/Controller/Lvl0/GRR (Granulate Remote)/helper/T_GRR_CTRL
TYPE T_GRR_CTRL :
STRUCT
	fbGrr: FB_GRR;
END_STRUCT
END_TYPE

// POUs/Controller/Lvl0/GRR (Granulate Remote)/helper/T_GRR_ID
TYPE T_GRR_ID :
STRUCT
	Grr: INT;
END_STRUCT
END_TYPE

// POUs/Controller/Lvl0/GRR (Granulate Remote)/helper/T_GRR_IO
TYPE T_GRR_IO :
STRUCT
	Out_intCommand: REFERENCE TO INT;
	Out_intConveyorBelt: REFERENCE TO INT;
	Out_intPowderVibrator: REFERENCE TO INT;
	Out_intConveyorVibrator: REFERENCE TO INT;
	Out_intAnalogValue: REFERENCE TO INT;
	Out_uinFilterClearingCycleTime_min: REFERENCE TO UINT;
	Out_bolToggleBitGrr: REFERENCE TO BOOL;
	In_bolSystemOk: REFERENCE TO BOOL;
	In_bolMainPressureError: REFERENCE TO BOOL;
	In_bolEoffOrFuseOk: REFERENCE TO BOOL;
	In_bolPowderLowWarning: REFERENCE TO BOOL;
	In_bolAutoMode: REFERENCE TO BOOL;
	In_intState: REFERENCE TO INT;
	In_bolToggleBitGrn: REFERENCE TO BOOL;
	In_intMainPressure: REFERENCE TO INT;
END_STRUCT
END_TYPE

// POUs/Controller/Lvl0/GRR (Granulate Remote)/E_ALM_GRR
TYPE E_ALM_GRR :
(
	NONE := 1,
	SystemError := 2,
	MainPressureError := 3,
	EoffOrFuseError := 4,
	LowPowderWarning := 5,
	ManualOperation := 6,
	LostConnection := 7,
	MAX_E_ALM_GRR
) UINT;
END_TYPE

// POUs/Controller/Lvl0/GRR (Granulate Remote)/T_Ctrl_SIf_GRR
TYPE T_Ctrl_SIf_GRR :
STRUCT
	/// configuration
	Cfg: T_Ctrl_SIf_GRR_Cfg;
	/// parameter
	Par: T_Ctrl_SIf_GRR_Par;
	/// current values
	Cur: T_Ctrl_SIf_GRR_Cur;
	///io input
	In: T_Ctrl_SIf_GRR_In;
	///io output
	Out: T_Ctrl_SIf_GRR_Out;
	/// alarm number used in this controller
	Alm: ARRAY[1..(E_ALM_GRR.MAX_E_ALM_GRR - 1)] OF T_Ctrl_Alm;
END_STRUCT
END_TYPE

// POUs/Controller/Lvl0/GRR (Granulate Remote)/T_Ctrl_SIf_GRR_Cfg
TYPE T_Ctrl_SIf_GRR_Cfg :
STRUCT
	rMaxFreq_Hz: REAL;
END_STRUCT
END_TYPE

// POUs/Controller/Lvl0/GRR (Granulate Remote)/T_Ctrl_SIf_GRR_Cur
TYPE T_Ctrl_SIf_GRR_Cur :
STRUCT
	intMainPressure: INT;
END_STRUCT
END_TYPE

// POUs/Controller/Lvl0/GRR (Granulate Remote)/T_Ctrl_SIf_GRR_In
TYPE T_Ctrl_SIf_GRR_In :
STRUCT
	bolSystemOk				: T_Ctrl_IoBool;
	bolMainPressureError	: T_Ctrl_IoBool;
	bolEoffOrFuseOk			: T_Ctrl_IoBool;
	bolPowderLowWarning		: T_Ctrl_IoBool;
	bolAutoMode				: T_Ctrl_IoBool;
	intState				: T_Ctrl_IoInt;
	bolToggleBitGrn			: T_Ctrl_IoBool;
	intMainPressure			: T_Ctrl_IoInt;
END_STRUCT
END_TYPE

// POUs/Controller/Lvl0/GRR (Granulate Remote)/T_Ctrl_SIf_GRR_Out
TYPE T_Ctrl_SIf_GRR_Out :
STRUCT
	intCommand						: BASE_PLC.T_Ctrl_IoInt;
	intConveyorBelt					: T_Ctrl_IoInt;
	intPowderVibrator				: T_Ctrl_IoInt;
	intConveyorVibrator				: T_Ctrl_IoInt;
	intAnalogValue					: T_Ctrl_IoInt;
	uinFilterClearingCycleTime_min	: T_Ctrl_IoUint;
	bolToggleBitGrr					: T_Ctrl_IoBool;
END_STRUCT
END_TYPE

// POUs/Controller/Lvl0/GRR (Granulate Remote)/T_Ctrl_SIf_GRR_Par
TYPE T_Ctrl_SIf_GRR_Par :
STRUCT
	rConveyorBelt_Hz: REAL;
	rPowderVibrator_Hz: REAL;
	rConveyorVibrator_Hz: REAL;
	rAnalogValue_p: REAL;
	uinFilterClearingCycleTime_min: UINT;
END_STRUCT
END_TYPE

// POUs/Controller/Lvl0/JCL (Jetter Client)/helper/T_JCL
TYPE T_JCL :
STRUCT
	io: T_JCL_IO;
	ctrl: T_JCL_CTRL;
	id: T_JCL_ID;
END_STRUCT
END_TYPE

// POUs/Controller/Lvl0/JCL (Jetter Client)/helper/T_JCL_CTRL
TYPE T_JCL_CTRL :
STRUCT
	fbJcl: FB_JCL;
	fbJcl_Tcp: FB_TCP;
END_STRUCT
END_TYPE

// POUs/Controller/Lvl0/JCL (Jetter Client)/helper/T_JCL_ID
TYPE T_JCL_ID :
STRUCT
	Jcl: INT;
	Jcl_Tcp: INT;
END_STRUCT
END_TYPE

// POUs/Controller/Lvl0/JCL (Jetter Client)/helper/T_JCL_IO
TYPE T_JCL_IO :
STRUCT
END_STRUCT
END_TYPE

// POUs/Controller/Lvl0/JCL (Jetter Client)/E_ALM_JCL
TYPE E_ALM_JCL :
(
	NONE := 1,
	JetterNotRun := 2,
	JetterManualWarning := 3,
	JetterManualError := 4,
	JetterEOff := 5,
	JetterCommunicationLost := 6,
	MAX_E_ALM_JCL
) UINT;
END_TYPE

// POUs/Controller/Lvl0/JCL (Jetter Client)/T_Ctrl_SIf_JCL
TYPE T_Ctrl_SIf_JCL :
STRUCT
	/// configuration
	Cfg: T_Ctrl_SIf_JCL_Cfg;
	/// parameter
	Par: T_Ctrl_SIf_JCL_Par;
	/// current values
	Cur: T_Ctrl_SIf_JCL_Cur;
	/// alarm number used in this controller
	Alm: ARRAY[1..(E_ALM_JCL.MAX_E_ALM_JCL - 1)] OF T_Ctrl_Alm;
END_STRUCT
END_TYPE

// POUs/Controller/Lvl0/JCL (Jetter Client)/T_Ctrl_SIf_JCL_Cfg
TYPE T_Ctrl_SIf_JCL_Cfg :
STRUCT
	/// FALSE = Do not allow manual mode, go to error if Jetter goes to manual / TRUE = Allow manual mode and stay in the last state 
	bolJetterManualModeAllowed: BOOL;
END_STRUCT
END_TYPE

// POUs/Controller/Lvl0/JCL (Jetter Client)/T_Ctrl_SIf_JCL_Cur
TYPE T_Ctrl_SIf_JCL_Cur :
STRUCT
	/// Additional states from TCP server
	/// Local control active. Commands from this client are ignored
	bolIsLocalControlled: BOOL;
	/// Remote control active. Commands from this client are accepted
	bolIsRemoteControlled: BOOL;
	/// Jetter ready for production
	bolReadyForProduction: BOOL;
	/// Print running, in production
	bolRunning: BOOL;
	/// System needs attention. Info or warning active
	bolNeedsAttention: BOOL;
	/// General error active
	bolError: BOOL;
	/// Cleaning cycle was aborted before finishing. Production not possible.
	bolCleaningIncomplete: BOOL;
	/// Print head needs cleaning.
	bolNeedsCleaning: BOOL;
	/// Timestamp of the last cleaning cycle. Format: YYYY-MM-DD-hh:mm:ss.xxx
	strDTOfLastCleaningCycle: STRING := '';
	/// Jetter state
	intJETState: INT;
END_STRUCT
END_TYPE

// POUs/Controller/Lvl0/JCL (Jetter Client)/T_Ctrl_SIf_JCL_Par
TYPE T_Ctrl_SIf_JCL_Par :
STRUCT
END_STRUCT
END_TYPE

// POUs/Controller/Lvl0/JCL (Jetter Client)/T_JCL_AlmMsg
TYPE T_JCL_AlmMsg :
STRUCT
	stHeader: ST_Header;
	/// Unique alarm number
	udiAlarmID: UDINT;
	/// Additional information
	udiInfo: UDINT;
	/// Corresponding alarm class
	usiClass: USINT;
	/// Corresponding controller ID
	uinCtrlID: UINT;
	/// Entry date and time
	strDTEntry: STRING(25);
	/// Alarm Text
	strText: STRING(255);
END_STRUCT
END_TYPE

// POUs/Controller/Lvl0/JCL (Jetter Client)/T_JCL_Command
{attribute 'pack_mode' := '1'}
TYPE T_JCL_Command :
STRUCT
	stHeader: ST_Header;
	usiCommand: USINT;
END_STRUCT
END_TYPE

// POUs/Controller/Lvl0/JCL (Jetter Client)/T_JCL_PrintDone
TYPE T_JCL_PrintDone :
STRUCT
	stHeader: ST_Header;
	usiBarcode: ARRAY[0..9] OF USINT;
	///  [%]
	usiInkLevelMainTank: USINT;
	///  [%]	
	usiInkLevelSupplyPrintModule1: USINT;
	///  [%]	
	usiInkLevelSupplyPrintModule2: USINT;
	///  [%]	
	usiInkLevelReturnPrintModule1: USINT;
	///  [%]	
	usiInkLevelReturnPrintModule2: USINT;
	///  [0.01 mbar]
	udiInkMeniscus: ARRAY[0..1] OF UDINT;
	///  [0.1 °C] 
	udiPrintHeadTemperature: ARRAY[0..1, 0..4] OF UDINT;
	///  [Micrometer]	//  Dimension of printed file calculated by DJM
	udiPrintWidthCalc: UDINT;
	///  [Micrometer]	//  Dimension of printed file calculated by DJM
	udiPrintLengthCalc: UDINT;
	///  [Micrometer]	//  Offset of print
	udiShiftXCalc: UDINT;
	///  [Micrometer]	//  Offset of print
	udiShiftYCalc: UDINT;
	///  [0.01°]		//  Offset of rotation angle 
	udiShiftAngleCalc: UDINT;
END_STRUCT
END_TYPE

// POUs/Controller/Lvl0/JCL (Jetter Client)/T_JCL_RequestCleaning
{attribute 'pack_mode' := '1'}
TYPE T_JCL_RequestCleaning :
STRUCT
	stHeader: ST_Header;
	/// Date and time of the last cleaning cycle
	strDTLastClean: STRING(25);
	/// Required interval for cleaning [min]
	uinRequiredInterval_min: UINT;
END_STRUCT
END_TYPE

// POUs/Controller/Lvl0/JCL (Jetter Client)/T_JCL_State
{attribute 'pack_mode' := '1'}
TYPE T_JCL_State :
STRUCT
	stHeader: ST_Header;
	usiMainState: USINT;
	///(Bit coded)	
	usiAddState: USINT;
END_STRUCT
END_TYPE

// POUs/Controller/Lvl0/JCL (Jetter Client)/U_JCL_Message
{attribute 'pack_mode' := '1'}
TYPE U_JCL_Message :

UNION
	Cmd: T_JCL_Command;
	State: T_JCL_State;
	PrintDone: T_JCL_PrintDone;
	ReqCleaning: T_JCL_RequestCleaning;
	AlmMsg: T_JCL_AlmMsg;
END_UNION

END_TYPE

// POUs/Controller/Lvl0/RAX(Rotative Axis)/E_ALM_RAX
{attribute 'qualified_only' := ''}
TYPE E_ALM_RAX :
(
	GeneralDrive := 1,
	GeneralNc,
	SwLimit,
	NegHwLimit,
	PosHwLimit,
	InterlockNegMove,
	InterlockPosMove,
	GeneralMCFUB,
	MAX_E_ALM
) UINT;
END_TYPE

// POUs/Controller/Lvl0/RAX(Rotative Axis)/T_Ctrl_SIf_RAX
TYPE T_Ctrl_SIf_RAX :
STRUCT
	///configuration
	Cfg: T_Ctrl_SIf_RAX_Cfg;
	///parameter
	Par: T_Ctrl_SIf_RAX_Par;
	///current values
	Cur: T_Ctrl_SIf_RAX_Cur;
	///alarm number used in this controller
	Alm: ARRAY[1..(E_ALM_RAX.MAX_E_ALM - 1)] OF T_Ctrl_Alm;
	///interlock of output/movements
	Ilk: T_Ctrl_SIf_RAX_Ilk;
END_STRUCT
END_TYPE

// POUs/Controller/Lvl0/RAX(Rotative Axis)/T_Ctrl_SIf_RAX_Cfg
TYPE T_Ctrl_SIf_RAX_Cfg :
STRUCT
	/// homing mode
	eHomingMode: MC_HomingMode;
	lreShortestWayWindow_deg: LREAL;
END_STRUCT
END_TYPE

// POUs/Controller/Lvl0/RAX(Rotative Axis)/T_Ctrl_SIf_RAX_Cur
TYPE T_Ctrl_SIf_RAX_Cur :
STRUCT
	/// [0.1°/s] current speed
	dinSpeed_0_1deg_s: DINT;
	/// [0.1°] current position
	dinPosition_0_1deg: DINT;
	/// [°] current modulo position
	dinModPosition_0_1deg: DINT;
	/// [0.1Nm] current torque
	dinTorque_0_1Nm: DINT;
	/// digital input1 from drive
	bol_di1: BOOL;
	/// digital input2 from drive
	bol_di2: BOOL;
	/// digital input3 from drive
	bol_di3: BOOL;
	/// digital input4 from drive
	bol_di4: BOOL;
	/// digital input5 from drive
	bol_di5: BOOL;
END_STRUCT
END_TYPE

// POUs/Controller/Lvl0/RAX(Rotative Axis)/T_Ctrl_SIf_RAX_Ilk
TYPE T_Ctrl_SIf_RAX_Ilk :
STRUCT
	/// interlock movment in positive direction
	bolMovePos: BOOL;
	/// interlock movment in negative direction
	bolMoveNeg: BOOL;
END_STRUCT
END_TYPE

// POUs/Controller/Lvl0/RAX(Rotative Axis)/T_Ctrl_SIf_RAX_Par
TYPE T_Ctrl_SIf_RAX_Par :
STRUCT
	/// [deg] home offset 
	dinHomeOffset_0_1deg: DINT;
	/// [0.1°] position init
	dinPositionInit_0_1deg: DINT;
	/// [0.1°] position absolute 
	dinPos_0_1deg: DINT;
	/// [0.1°] rel distance
	dinRelDist_0_1deg: DINT;
	/// [0.1°/s] position speed
	dinSpeed_0_1deg_s: DINT;
	///[%] percent from dinSetSpeed_0_1deg_s
	dinSpeed_per: DINT;
	/// [0.1°/s^2] position acceleration
	dintAccDec_0_1deg_s2: DINT;
	///[%] percent from dintAccDec_0_1deg_s2
	dinAcc_per: DINT;
	///[%] percent from dintAccDec_0_1deg_s2
	dinDec_per: DINT;
	/// [0.1°/s^2] position deceleration fast em stop
	dinSetDecFast_0_1deg_s2: DINT;
	/// [0.1°] negative sw limite
	dinSWLimitNeg_0_1deg: DINT;
	/// [0.1°] positive sw limite
	dinSWLimitPos_0_1deg: DINT;
END_STRUCT
END_TYPE

// POUs/Controller/Lvl1/BCH (Barcode with DataChannel)/helper/T_BCH
TYPE T_BCH :
STRUCT
	io: T_BCH_IO;
	ctrl: T_BCH_CTRL;
	id: T_BCH_ID;
	datachn: T_BCH_DATACHN;
END_STRUCT
END_TYPE

// POUs/Controller/Lvl1/BCH (Barcode with DataChannel)/helper/T_BCH_CTRL
TYPE T_BCH_CTRL :
STRUCT
	fbBch: FB_BCH;
	fbBch_Bcc: FB_BCC;
	fbBch_Bcc_Bcd: FB_BCD;
END_STRUCT
END_TYPE

// POUs/Controller/Lvl1/BCH (Barcode with DataChannel)/helper/T_BCH_DATACHN
TYPE T_BCH_DATACHN :
STRUCT
	rSendData: T_IdBaseSendData;
END_STRUCT
END_TYPE

// POUs/Controller/Lvl1/BCH (Barcode with DataChannel)/helper/T_BCH_ID
TYPE T_BCH_ID :
STRUCT
	Bch: INT;
	Bch_Bcc: INT;
	Bch_Bcc_Bcd: INT;
END_STRUCT
END_TYPE

// POUs/Controller/Lvl1/BCH (Barcode with DataChannel)/helper/T_BCH_IO
TYPE T_BCH_IO :
STRUCT
	In_bolSensorTrigScan: REFERENCE TO BOOL;
END_STRUCT
END_TYPE

// POUs/Controller/Lvl1/BCH (Barcode with DataChannel)/E_ALM_BCH
TYPE E_ALM_BCH :
(
	DataChannelMissing := 1,
	DataChannelBufferFull,
	BarcodeNotReadCorrectly,
	MAX_E_ALM_BCH
) UINT;
END_TYPE

// POUs/Controller/Lvl1/BCH (Barcode with DataChannel)/T_Ctrl_SIf_BCH
TYPE T_Ctrl_SIf_BCH :
STRUCT
	/// configuration
	Cfg: T_Ctrl_SIf_BCH_Cfg;
	/// parameter
	Par: T_Ctrl_SIf_BCH_Par;
	/// current values
	Cur: T_Ctrl_SIf_BCH_Cur;
	/// Input layer
	In: T_Ctrl_SIf_BCH_In;
	/// alarm number used in this controller
	Alm: ARRAY[1..(E_ALM_BCH.MAX_E_ALM_BCH - 1)] OF T_Ctrl_Alm;
END_STRUCT
END_TYPE

// POUs/Controller/Lvl1/BCH (Barcode with DataChannel)/T_Ctrl_SIf_BCH_Cfg
TYPE T_Ctrl_SIf_BCH_Cfg :
STRUCT
	/// TRUE = Enable Data Channel; False = Disable DataChannel
	bolEnableDataChannel			: BOOL;
	// TRUE = Negative Trigger Signal, FALSE = Positive Trigger Signal
	bolNegativeTriggerSignal 		: BOOL;
END_STRUCT
END_TYPE

// POUs/Controller/Lvl1/BCH (Barcode with DataChannel)/T_Ctrl_SIf_BCH_Cur
TYPE T_Ctrl_SIf_BCH_Cur :
STRUCT
END_STRUCT
END_TYPE

// POUs/Controller/Lvl1/BCH (Barcode with DataChannel)/T_Ctrl_SIf_BCH_In
TYPE T_Ctrl_SIf_BCH_In :
STRUCT
	/// Trigger the measurement sensor
	bolSensorTrigScan: BASE_PLC.T_Ctrl_IoBool;
END_STRUCT
END_TYPE

// POUs/Controller/Lvl1/BCH (Barcode with DataChannel)/T_Ctrl_SIf_BCH_Par
TYPE T_Ctrl_SIf_BCH_Par :
STRUCT
END_STRUCT
END_TYPE

// POUs/Controller/Lvl1/MDC [Malteser Drive Controller]/E_ALM_MDC
TYPE E_ALM_MDC :
(
	TableSensorTimeout 		:= 1,
	CrossSensorTimeout		:= 2,
	PositionSame			:= 3,
	MAX_E_ALM_MDC
);
END_TYPE

// POUs/Controller/Lvl1/MDC [Malteser Drive Controller]/T_Ctrl_SIf_MDC
TYPE T_Ctrl_SIf_MDC :
STRUCT
	///configuration
	Cfg: T_Ctrl_SIf_MDC_Cfg;
	///parameter
	Par: T_Ctrl_SIf_MDC_Par;
	///current values
	Cur: T_Ctrl_SIf_MDC_Cur;
	///io input
	In: T_Ctrl_SIf_MDC_In;
	///io output
	Out: T_Ctrl_SIf_MDC_Out;
	///alarm number used in this controller
	Alm: ARRAY[1..MAX_E_ALM_MDC] OF T_Ctrl_Alm;
	///interlock of output/movements
	Ilk: T_Ctrl_SIf_MDC_Ilk;
END_STRUCT
END_TYPE

// POUs/Controller/Lvl1/MDC [Malteser Drive Controller]/T_Ctrl_SIf_MDC_Cfg
TYPE T_Ctrl_SIf_MDC_Cfg :
STRUCT
	/// Number of positions in 360° of the Malteser drive
	uintPositionPerTurn		: UINT;
END_STRUCT
END_TYPE

// POUs/Controller/Lvl1/MDC [Malteser Drive Controller]/T_Ctrl_SIf_MDC_Cur
TYPE T_Ctrl_SIf_MDC_Cur :
STRUCT	
	/// Actual Position as position 
	uintActualPosition			: UINT;
	/// actual turning direction
	eActualTurningDirection		: E_TURN_DIRECTION;
	/// Reference still ok
	bolReferenceOk				: BOOL;		
END_STRUCT
END_TYPE

// POUs/Controller/Lvl1/MDC [Malteser Drive Controller]/T_Ctrl_SIf_MDC_Ilk
TYPE T_Ctrl_SIf_MDC_Ilk :
STRUCT
END_STRUCT
END_TYPE

// POUs/Controller/Lvl1/MDC [Malteser Drive Controller]/T_Ctrl_SIf_MDC_In
TYPE T_Ctrl_SIf_MDC_In :
STRUCT
	/// Is the cross in sensor positinon. One rotation step done.
	bolCrossPositionSensor				: BASE_PLC.T_Ctrl_IoBool;
	/// Is the table at 0° degrees
	bolTablePositionSensor				: BASE_PLC.T_Ctrl_IoBool;
END_STRUCT
END_TYPE

// POUs/Controller/Lvl1/MDC [Malteser Drive Controller]/T_Ctrl_SIf_MDC_Out
TYPE T_Ctrl_SIf_MDC_Out :
STRUCT
	intActualPosition		: BASE_PLC.T_Ctrl_IoInt;
END_STRUCT
END_TYPE

// POUs/Controller/Lvl1/MDC [Malteser Drive Controller]/T_Ctrl_SIf_MDC_Par
TYPE T_Ctrl_SIf_MDC_Par :
STRUCT
	/// <0 = Turn left; =0 automatic; >0 turn right
	intTurnDirection					: INT;
	/// Position to go to if comand turn is given. 0 = initialization position
	uinPositionToGo						: UINT;
	/// [ms] time to rotate one step 
	udiStepRotationTime_ms				: UDINT;
	/// [ms] initialization timeout time
	udiInitializationTime_ms			: UDINT;
	/// [ms] simulation time to rotate one step
	udiSimStepRotationTime_ms			: UDINT;
	/// [ms] simulation initialization timeout time
	udiSimInitializationTime_ms			: UDINT;
	/// [ms] simulation time to start rotate and Cross sensor needs to go away
	udiSimStartRotationTime_ms			: UDINT;
	/// [rpm] PrePosition Speed
	uinPrePositionSpeed_rpm				: UINT;
	/// [rpm] Position Speed
	uinPositionSpeed_rpm				: UINT;
END_STRUCT
END_TYPE

// POUs/Controller/Lvl1/OVN (Oven)/helper/T_OVN
TYPE T_OVN :
STRUCT
	io		: T_OVN_IO;
	ctrl	: T_OVN_CTRL;
	id		: T_OVN_ID;
	datachn	: T_OVN_DATACHN;
END_STRUCT
END_TYPE

// POUs/Controller/Lvl1/OVN (Oven)/helper/T_OVN_CTRL
TYPE T_OVN_CTRL :
STRUCT
	fbOvn: FB_OVN;
	fbOvn_Ibh: FB_IBH;
END_STRUCT
END_TYPE

// POUs/Controller/Lvl1/OVN (Oven)/helper/T_OVN_DATACHN
TYPE T_OVN_DATACHN :
STRUCT
	rSendData	: T_OvenSendData;
END_STRUCT
END_TYPE

// POUs/Controller/Lvl1/OVN (Oven)/helper/T_OVN_ID
TYPE T_OVN_ID :
STRUCT
	Ovn: INT;
	Ovn_Ibh: INT;
END_STRUCT
END_TYPE

// POUs/Controller/Lvl1/OVN (Oven)/helper/T_OVN_IO
TYPE T_OVN_IO :
STRUCT
	Out_uinBcrOvenAEvent: REFERENCE TO UINT;
	Out_udiBcrOvenACode: REFERENCE TO ULINT;
	Out_uinBcrOvenBEvent: REFERENCE TO UINT;
	Out_udiBcrOvenBCode: REFERENCE TO ULINT;
	In_bolBcrDistributionTrigger: REFERENCE TO BOOL;
	In_udiBarcode_new_1: REFERENCE TO ULINT;
	In_udiBarcode_new_2: REFERENCE TO ULINT;
	In_uinNew_element_1: REFERENCE TO UINT;
	In_uinNew_element_2: REFERENCE TO UINT;
	In_udiBarcode_delete_1: REFERENCE TO ULINT;
	In_udiBarcode_delete_2: REFERENCE TO ULINT;
	In_uinDelete_element_1: REFERENCE TO UINT;
	In_uinDelete_element_2: REFERENCE TO UINT;
END_STRUCT
END_TYPE

// POUs/Controller/Lvl1/OVN (Oven)/E_ALM_OVN
TYPE E_ALM_OVN :
(
	NONE := 0,
	TempError := 1,
	AirError := 2,
	SpeedError := 3,
	TimeoutError := 4,
	ParameterWarning := 5,
	ConnectionError := 6,
	WrongMode := 7,
	/// OvertemperaturePowerSection						- software reset	- operating mode must be reelected
	Tesoma10000 := 8,
	/// FailureOfActiveCoolingUnit
	Tesoma10002 := 9,
	/// ActiveCoolingUnitNotRunning
	Tesoma10003 := 10,
	/// FailureFuseGeneral													- transport starts immediately when sensor is free
	Tesoma10006 := 11,
	/// BeltPositionControlSensorError					- software reset
	Tesoma10010 := 12,
	/// BeltEdgeShutOff									- software reset
	Tesoma10011 := 13,
	/// FaultBeltSpeed									- software reset
	Tesoma10012 := 14,
	/// TransportOverload
	Tesoma10013 := 15,
	/// BeltControlDeviceFault							- software reset	- reset FC
	Tesoma10014 := 16,
	/// EmergencyStop														- would be resettable, but since power is gone, the acknowledge does not arrive
	Tesoma10016 := 17,
	/// BeltWearMonitor
	Tesoma10023 := 18,
	/// ControlCabinetFan
	Tesoma10024 := 19,
	/// ControlCabinetTemperatureTooHigh
	Tesoma10025 := 20,
	/// PowerSupplyFailure
	Tesoma10026 := 21,
	/// IntakeHoodTemperatureExceeded
	Tesoma10027 := 22,
	/// AirPressureTooLow
	Tesoma10030 := 23,
	/// BeltPositionControlNotWorking
	Tesoma10031 := 24,
	/// ErrorCoolingDeviceControlCabinet
	Tesoma10032 := 25,
	/// ControlCabinetCoolerAndSmallDrivesFuseFailure
	Tesoma10034 := 26,
	/// LimitSwitchingOff								- software reset	- after elimination, reactivates according zone
	Tesoma10x00 := 27,
	/// OvertemperatureStl								- software reset	- after elimination AND reset, the STL reactivates the accordant zone
	Tesoma10x01 := 28,
	/// FuseTriggered									- software reset	- after elimination, reactivates the accordant zone
	Tesoma10x02 := 29,
	/// FailureExhaustAirDps								- software reset	- after elimination, reactivates the accordant zone
	Tesoma10x03 := 30,
	/// ErrorFrequencyConverter							- software reset	- after elimination AND reset, the FC reactivates the accordant zone
	Tesoma10x07 := 31,
	/// TemperatureSensorIrDefective
	Tesoma10x13 := 32,
	/// FaultFrameCoolingSystemDps
	Tesoma10x14 := 33,
	/// FaultExhaustAirDps
	Tesoma10x15 := 34,
	/// TemperatureFault									- software reset
	Tesoma13x00 := 35,
	TesomaUnknown := 36,
	HostConnectionLost := 37,
	SettingsChanged := 38,
	MAX_E_ALM_OVN
);
END_TYPE

// POUs/Controller/Lvl1/OVN (Oven)/T_Ctrl_SIf_OVN
TYPE T_Ctrl_SIf_OVN :
STRUCT
	///configuration
	Cfg: T_Ctrl_SIf_OVN_Cfg;
	///parameter
	Par: T_Ctrl_SIf_OVN_Par;
	///current values
	Cur: T_Ctrl_SIf_OVN_Cur;
	///io input
	In: T_Ctrl_SIf_OVN_In;
	///io output
	Out: T_Ctrl_SIf_OVN_Out;
	///alarm number used in this controller
	Alm: ARRAY[1..(E_ALM_OVN.MAX_E_ALM_OVN - 1)] OF T_Ctrl_Alm;
END_STRUCT
END_TYPE

// POUs/Controller/Lvl1/OVN (Oven)/T_Ctrl_SIf_OVN_Cfg
TYPE T_Ctrl_SIf_OVN_Cfg EXTENDS T_Ctrl_SIf_MOD_Cfg :
STRUCT
	/// Number of Modules in use 
	uiNumberOfModules: UINT;
	/// Length of one Module 
	diModuleLength_mm: DINT;
	/// Distance before the first Module 
	diDistanceBeforeOven_mm: DINT;
	/// Distance after the last Module 
	diDistanceAfterOven_mm: DINT;
	/// Maximal Belt Speed in mm/min 
	diMaxSpeed_mm_min: DINT;
	/// Minimal Belt Speed in mm/min 
	diMinSpeed_mm_min: DINT;
	/// Minimal Temperature in deci °C 
	diMinTemp_dc: DINT;
	/// Maximal Temperature in deci °C 
	diMaxTemp_dc: DINT;
	/// Minimal Airflow in % 
	diMinAir_p: DINT;
	/// Maximal Airflow in % 
	diMaxAir_p: DINT;
	/// Auto Continue After Connection Error
	bAutoContinueAfterConnectionError: BOOL;
	/// Enable Data Channel
	bolDataChannelEnable: BOOL;
	/// ignore waiting for Paper to eject in OFFBusy
	bIgnoreOffBusyWaitPaper: BOOL;
END_STRUCT
END_TYPE

// POUs/Controller/Lvl1/OVN (Oven)/T_Ctrl_SIf_OVN_Cur
TYPE T_Ctrl_SIf_OVN_Cur EXTENDS T_Ctrl_SIf_MOD_Cur :
STRUCT
	/// Belt Speed in mm/min 
	diSpeed_mm_min: DINT;
	/// Temperature in deci °C 
	adiTemp_dc: ARRAY[0..(MAX_NUMBER_OF_OVEN_MODULES - 1)] OF DINT;
	/// Airflow in % 
	adiAir_p: ARRAY[0..(MAX_NUMBER_OF_OVEN_MODULES - 1)] OF DINT;
END_STRUCT
END_TYPE

// POUs/Controller/Lvl1/OVN (Oven)/T_Ctrl_SIf_OVN_In
TYPE T_Ctrl_SIf_OVN_In :
STRUCT
END_STRUCT
END_TYPE

// POUs/Controller/Lvl1/OVN (Oven)/T_Ctrl_SIf_OVN_Out
TYPE T_Ctrl_SIf_OVN_Out :
STRUCT
END_STRUCT
END_TYPE

// POUs/Controller/Lvl1/OVN (Oven)/T_Ctrl_SIf_OVN_Par
TYPE T_Ctrl_SIf_OVN_Par EXTENDS T_Ctrl_SIf_MOD_Par :
STRUCT
	/// Belt Speed in mm/min 
	diSpeed_mm_min: DINT;
	/// Belt Speed Band in mm/min 
	diSpeedBand1_mm_min: DINT;
	/// Belt Speed Band in mm/min 
	diSpeedBand2_mm_min: DINT;
	/// Belt Speed Timeout in ms 
	udiSpeedTimeout_ms: UDINT;
	/// Temperature in deci °C 
	adiTemp_dc: ARRAY[0..(MAX_NUMBER_OF_OVEN_MODULES - 1)] OF DINT;
	/// Temperature Band in deci °C 
	adiTempBand1_dc: ARRAY[0..(MAX_NUMBER_OF_OVEN_MODULES - 1)] OF DINT;
	/// Temperature Band in deci °C 
	adiTempBand2_dc: ARRAY[0..(MAX_NUMBER_OF_OVEN_MODULES - 1)] OF DINT;
	/// Temperature Timeout in ms 
	audiTempTimeout_ms: ARRAY[0..(MAX_NUMBER_OF_OVEN_MODULES - 1)] OF UDINT;
	/// Airflow in % 
	adiAir_p: ARRAY[0..(MAX_NUMBER_OF_OVEN_MODULES - 1)] OF DINT;
	/// Airflow Band in % 
	adiAirBand1_p: ARRAY[0..(MAX_NUMBER_OF_OVEN_MODULES - 1)] OF DINT;
	/// Airflow Band in % 
	adiAirBand2_p: ARRAY[0..(MAX_NUMBER_OF_OVEN_MODULES - 1)] OF DINT;
	/// Airflow Timeout in ms 
	audiAirTimeout_ms: ARRAY[0..(MAX_NUMBER_OF_OVEN_MODULES - 1)] OF UDINT;
	udiTimeoutOffBusy_ms: UDINT;
	udiTimeoutRunBusyReaction_ms: UDINT;
	udiTimeoutRunBusyInBand_ms: UDINT;
	udiTimeoutBeltOnlyReaction_ms: UDINT;
	udiTimeoutBeltOnlyBusy_ms: UDINT;
END_STRUCT
END_TYPE

// POUs/Controller/Lvl1/OVN (Oven)/T_Data
{attribute 'enable_dynamic_creation' := ''}
TYPE T_Data :
STRUCT
	uliBarcode: ULINT;
	bTrash: BOOL;
	diDistance_um: DINT;
	diSumTemp_mc: ARRAY[0..(MAX_NUMBER_OF_OVEN_MODULES - 1)] OF DINT;
	diCyclesInModule: ARRAY[0..(MAX_NUMBER_OF_OVEN_MODULES - 1)] OF DINT;
	bBarcodeMissed: BOOL;
END_STRUCT
END_TYPE

// POUs/Controller/Lvl1/PTA [Paper Transport Alignment]/helper/T_PTA
TYPE T_PTA :
STRUCT
	io:		T_PTA_IO;
	ctrl:	T_PTA_CTRL;
	id:		T_PTA_ID;
END_STRUCT
END_TYPE

// POUs/Controller/Lvl1/PTA [Paper Transport Alignment]/helper/T_PTA_CTRL
TYPE T_PTA_CTRL :
STRUCT
	fbPta: FB_PTB;	// PTA is a special type of PTB
	fbPta_Umc: FB_UMC;
END_STRUCT
END_TYPE

// POUs/Controller/Lvl1/PTA [Paper Transport Alignment]/helper/T_PTA_ID
TYPE T_PTA_ID :
STRUCT
	Pta: INT;
	Pta_Umc: INT;
END_STRUCT
END_TYPE

// POUs/Controller/Lvl1/PTA [Paper Transport Alignment]/helper/T_PTA_IO
TYPE T_PTA_IO :
STRUCT
	In_bolInputSensor: REFERENCE TO BOOL;
	In_bolOutputSensor: REFERENCE TO BOOL;
	
	In_uinUmc_Status: REFERENCE TO UINT;
	In_uinUmc_ActualSpeed: REFERENCE TO UINT;
	In_uinUmc_SetSpeed: REFERENCE TO UINT;
	In_uinUmc_IOData1: REFERENCE TO WORD;
	In_uinUmc_ECatState: REFERENCE TO UINT;
	In_strUmc_ECatNetId: REFERENCE TO AMSNETID;
	In_uinUmc_ECatPort: REFERENCE TO WORD;
	Out_uinUmc_Control: REFERENCE TO UINT;
	Out_uinUmc_SetSpeed: REFERENCE TO UINT;
END_STRUCT
END_TYPE

// POUs/Controller/Lvl1/PTB [Paper Transport Belt]/BeltParameterFunction/T_Belt_Cfg_Base
TYPE T_Belt_Cfg_Base :
STRUCT
	/// Assign the motor rotation to a belt direction.
	intForwardDirection				: INT;
	/// Assign the motor rotation to a belt direction.
	intBackwardDirection			: INT;
	/// [mm] the belt travels per motor rotation
	reaRpmDistance_mm					: REAL;
END_STRUCT
END_TYPE

// POUs/Controller/Lvl1/PTB [Paper Transport Belt]/BeltParameterFunction/T_Belt_Cur_Base
TYPE T_Belt_Cur_Base :
STRUCT
	/// [mm/s] Belt speed
	uinBeltSpeed_mms						: UINT;
	/// [rpm] Belt speed
	uinBeltSpeed_rpm						: UINT;
END_STRUCT
END_TYPE

// POUs/Controller/Lvl1/PTB [Paper Transport Belt]/BeltParameterFunction/T_Belt_Par_Base
TYPE T_Belt_Par_Base :
STRUCT
	/// eSpeedControlSelection.EFFECTIVE_SPEED : [mm/sec] Target speed. Uses reaRpmDistance_mm and uinLC11 to calculate the rpm
	uinBeltSpeed						: UINT;
	/// eSpeedControlSelection.EFFECTIVE_SPEED : [mm/sec] Target speed. Uses reaRpmDistance_mm and uinLC11 to calculate the rpm
	uinStackSpeed						: UINT;
END_STRUCT
END_TYPE

// POUs/Controller/Lvl1/PTB [Paper Transport Belt]/helper/T_PTB
TYPE T_PTB :
STRUCT
	io:		T_PTB_IO;
	ctrl:	T_PTB_CTRL;
	id:		T_PTB_ID;
END_STRUCT
END_TYPE

// POUs/Controller/Lvl1/PTB [Paper Transport Belt]/helper/T_PTB_CTRL
TYPE T_PTB_CTRL :
STRUCT
	fbPtb: FB_PTB;
	fbPtb_Umc: FB_UMC;
	fbPtb_Vpc: FB_VPC;
END_STRUCT
END_TYPE

// POUs/Controller/Lvl1/PTB [Paper Transport Belt]/helper/T_PTB_ID
TYPE T_PTB_ID :
STRUCT
	Ptb: INT;
	Ptb_Umc: INT;
	Ptb_Vpc: INT;
END_STRUCT
END_TYPE

// POUs/Controller/Lvl1/PTB [Paper Transport Belt]/helper/T_PTB_IO
TYPE T_PTB_IO :
STRUCT
	In_bolInputSensor: REFERENCE TO BOOL;
	In_bolOutputSensor: REFERENCE TO BOOL;
	
	In_bolVpc_VacuumSensor: REFERENCE TO BOOL;
	In_bolVpc_PumpOk: REFERENCE TO BOOL;
	Out_bolVpc_PumpOn: REFERENCE TO BOOL;	

	In_bolUmc_EmoOk: REFERENCE TO BOOL;
	In_uinUmc_Status: REFERENCE TO UINT;
	In_uinUmc_ActualSpeed: REFERENCE TO UINT;
	In_uinUmc_SetSpeed: REFERENCE TO UINT;
	In_uinUmc_IOData1: REFERENCE TO WORD;
	In_uinUmc_ECatState: REFERENCE TO UINT;
	In_strUmc_ECatNetId: REFERENCE TO AMSNETID;
	In_uinUmc_ECatPort: REFERENCE TO WORD;
	Out_uinUmc_Control: REFERENCE TO UINT;
	Out_uinUmc_SetSpeed: REFERENCE TO UINT;
END_STRUCT
END_TYPE

// POUs/Controller/Lvl1/PTB [Paper Transport Belt]/E_ALM_PTB
TYPE E_ALM_PTB :
(
	TestAlarm := 1,
	MAX_E_ALM_PTB 
);
END_TYPE

// POUs/Controller/Lvl1/PTB [Paper Transport Belt]/E_BELT_DIRECTION
TYPE E_BELT_DIRECTION :
(
	FORWARD			:= 0,
	BACKWARD		:= 1,
	MAX_E_BELT_DIRECTION
);
END_TYPE

// POUs/Controller/Lvl1/PTB [Paper Transport Belt]/E_PTB_MODE
TYPE E_PTB_MODE :
(
	Endless	,		// 0
	ToSensor,		// 1
	ToDistance,		// 2
	ToTime,			// 3
	Stack,			// 4
	MAX_E_PTB_MODE
);
END_TYPE

// POUs/Controller/Lvl1/PTB [Paper Transport Belt]/E_PTB_PaperDirection
TYPE E_PTB_PaperDirection :
(
	Portrait,
	Landscape,
	MAX_E_PTB_PaperDirection
);
END_TYPE

// POUs/Controller/Lvl1/PTB [Paper Transport Belt]/T_Ctrl_SIf_PTB
TYPE T_Ctrl_SIf_PTB :
STRUCT
	///configuration
	Cfg: T_Ctrl_SIf_PTB_Cfg;
	///parameter
	Par: T_Ctrl_SIf_PTB_Par;
	///current values
	Cur: T_Ctrl_SIf_PTB_Cur;
	///io input
	In: T_Ctrl_SIf_PTB_In;
	///io output
	Out: T_Ctrl_SIf_PTB_Out;
	///alarm number used in this controller
	Alm: ARRAY[1..E_ALM_PTB.MAX_E_ALM_PTB] OF T_Ctrl_Alm;
	///interlock of output/movements
	Ilk: T_Ctrl_SIf_PTB_Ilk;
END_STRUCT
END_TYPE

// POUs/Controller/Lvl1/PTB [Paper Transport Belt]/T_Ctrl_SIf_PTB_Cfg
TYPE T_Ctrl_SIf_PTB_Cfg :
STRUCT
	// Function Mode
	eMode							: E_PTB_MODE;
	// Vacuum pump present
	bolVacuumPresent				: BOOL;
	// [mm] Length of the belt
	udiBeltLength_mm				: UDINT;
	// Belt Parameter	
	rBeltParam						: T_Belt_Cfg_Base;
	// Enable Entry Belt Sensor Debounce
	bolEntrySensorDebounceEnable	: BOOL;
	// Enable Exit Belt Sensor Debounce
	bolExitSensorDebounceEnable		: BOOL;
END_STRUCT
END_TYPE

// POUs/Controller/Lvl1/PTB [Paper Transport Belt]/T_Ctrl_SIf_PTB_Cur
	TYPE T_Ctrl_SIf_PTB_Cur :
STRUCT	
	/// actual belt direction
	eActualDirection						: E_BELT_DIRECTION;
	/// [mm] Distance to move if Move Mode is distance
	udiDistanceToMove_mm					: UDINT;
	/// [ms] Time to move
	udiTimeToMove_ms						: UDINT;
	// Belt parameter
	rBeltParam								: T_Belt_Cur_Base;
	// Belt Run Time
	udiBeltTimeBase_mm						: UDINT;
	// Paper on the belt
	uinPaperOnBelt							: UINT;
	// Pointer to the Position list of the paper on the belt
	pPositionList							: POINTER TO T_PTR_STRUCT;
END_STRUCT
END_TYPE

// POUs/Controller/Lvl1/PTB [Paper Transport Belt]/T_Ctrl_SIf_PTB_Ilk
TYPE T_Ctrl_SIf_PTB_Ilk :
STRUCT
END_STRUCT
END_TYPE

// POUs/Controller/Lvl1/PTB [Paper Transport Belt]/T_Ctrl_SIf_PTB_In
TYPE T_Ctrl_SIf_PTB_In :
STRUCT
	bolBeltEntrySensor			: BASE_PLC.T_Ctrl_IoBool;
	bolBeltExitSensor			: BASE_PLC.T_Ctrl_IoBool;
	bolBeltEntrySensorPEdge		: BASE_PLC.T_Ctrl_IoBool;
	bolBeltEntrySensorNEdge		: BASE_PLC.T_Ctrl_IoBool;
	bolBeltExitSensorPEdge		: BASE_PLC.T_Ctrl_IoBool;
	bolBeltExitSensorNEdge		: BASE_PLC.T_Ctrl_IoBool;
END_STRUCT
END_TYPE

// POUs/Controller/Lvl1/PTB [Paper Transport Belt]/T_Ctrl_SIf_PTB_Out
TYPE T_Ctrl_SIf_PTB_Out :
STRUCT

END_STRUCT
END_TYPE

// POUs/Controller/Lvl1/PTB [Paper Transport Belt]/T_Ctrl_SIf_PTB_Par
TYPE T_Ctrl_SIf_PTB_Par :
STRUCT
	/// <0 = Backward; =0 None; >0 forward
	intDirection						: INT;
	/// [mm] Distance to move if Move Mode is distance
	udiDistanceToMove_mm				: UDINT;
	/// [ms] Time to move
	udiTimeToMove_ms					: UDINT;
	/// Stack hight in # of sheets
	uinPaperStackHight					: UINT;
	/// Automatic ejecting the paper if stackhight is reached
	bolAutoEjectAfterStack				: BOOL;
	/// Automatic stacking the paper after ejecting all paper
	bolAutoStackAfterEject				: BOOL;
	/// Belt Parameter
	rBeltParam							: T_Belt_Par_Base;
	// [ms] Stack delay time - Delay before out motor can move after paper entered system
	udiStackDelayTime_ms				: UDINT;
	// [mm] Belt Length
	udiBeltLength_mm					: UDINT;
	// Page running format
	ePaperOrientation					: E_PTB_PaperDirection;
	/// [mm] Paper Hight
	uinPaperHight_mm					: UINT;
	/// [mm] Paper Width
	uinPaperWidth_mm					: UINT;
	// [ms] Input Parameter Debounce time
	uinInputSignalDebounceTime_ms		: UINT;
END_STRUCT
END_TYPE

// POUs/Controller/Lvl2/PBC [Paper Buffer Controller]/helper/T_PBC
TYPE T_PBC :
STRUCT
	io: T_PBC_IO;
	ctrl: T_PBC_CTRL;
	id: T_PBC_ID;
END_STRUCT
END_TYPE

// POUs/Controller/Lvl2/PBC [Paper Buffer Controller]/helper/T_PBC_CTRL
TYPE T_PBC_CTRL :
STRUCT
	fbPbc_PtbDeStacker: FB_PTB;
	fbPbc_PtbDeStacker_Umc: FB_UMC;
	fbPbc_PtbBelt: FB_PTB;
	fbPbc_PtbBelt_Umc: FB_UMC;
	fbPbc_PtbBelt_Vpc: FB_VPC;
	fbPbc: FB_PBC;
END_STRUCT
END_TYPE

// POUs/Controller/Lvl2/PBC [Paper Buffer Controller]/helper/T_PBC_ID
TYPE T_PBC_ID :
STRUCT
	Pbc: INT;
	Pbc_PtbDeStacker: INT;
	Pbc_PtbDeStacker_Umc: INT;
	Pbc_PtbBelt: INT;
	Pbc_PtbBelt_Umc: INT;
	Pbc_PtbBelt_Vpc: INT;
END_STRUCT
END_TYPE

// POUs/Controller/Lvl2/PBC [Paper Buffer Controller]/helper/T_PBC_IO
TYPE T_PBC_IO :
STRUCT
	///TODO: describe why this is here
	In_bolPts_PaperSensor: REFERENCE TO BOOL;
	In_bolInputSensor: REFERENCE TO BOOL;
	In_bolOutputSensor: REFERENCE TO BOOL;
	In_bolCapacitySensor: REFERENCE TO BOOL;
	In_bolDoublePaperSensor: REFERENCE TO BOOL;
	In_bolAirPressureOk: REFERENCE TO BOOL;
	Out_bolAirPressureOn: REFERENCE TO BOOL;

	In_bolPtbBelt_Vpc_VacuumSensor: REFERENCE TO BOOL;
	In_bolPtbBelt_Vpc_PumpOk: REFERENCE TO BOOL;
	Out_bolPtbBelt_Vpc_PumpOn: REFERENCE TO BOOL;

	In_uinPtbBelt_Umc_Status: REFERENCE TO UINT;
	In_uinPtbBelt_Umc_ActualSpeed: REFERENCE TO UINT;
	In_uinPtbBelt_Umc_SetSpeed: REFERENCE TO UINT;
	In_uinPtbBelt_Umc_IOData1: REFERENCE TO WORD;
	In_uinPtbBelt_Umc_ECatState: REFERENCE TO UINT;
	In_strPtbBelt_Umc_ECatNetId: REFERENCE TO AMSNETID;
	In_uinPtbBelt_Umc_ECatPort: REFERENCE TO WORD;
	Out_uinPtbBelt_Umc_Control: REFERENCE TO UINT;
	Out_uinPtbBelt_Umc_SetSpeed: REFERENCE TO UINT;

	In_uinPtbDeStacker_Umc_Status: REFERENCE TO UINT;
	In_uinPtbDeStacker_Umc_ActualSpeed: REFERENCE TO UINT;
	In_uinPtbDeStacker_Umc_SetSpeed: REFERENCE TO UINT;
	In_uinPtbDeStacker_Umc_IOData1: REFERENCE TO WORD;
	In_uinPtbDeStacker_Umc_ECatState: REFERENCE TO UINT;
	In_strPtbDeStacker_Umc_ECatNetId: REFERENCE TO AMSNETID;
	In_uinPtbDeStacker_Umc_ECatPort: REFERENCE TO WORD;
	Out_uinPtbDeStacker_Umc_Control: REFERENCE TO UINT;
	Out_uinPtbDeStacker_Umc_SetSpeed: REFERENCE TO UINT;
END_STRUCT
END_TYPE

// POUs/Controller/Lvl2/PBC [Paper Buffer Controller]/E_ALM_PBC
TYPE E_ALM_PBC :
(
	PaperTransport := 1,
	BufferFull := 2,
	BufferEmpty := 3,
	DoublePaperError := 4,
	DataChannelBufferFull := 5,
	DataChannelSend := 6,
	PaperInject := 7,
	PaperInjectRetry := 8,
	DoNotReleaseItems := 9,
	DoublePaperWarning := 10,
	MAX_E_ALM_PBC
);
END_TYPE

// POUs/Controller/Lvl2/PBC [Paper Buffer Controller]/T_Ctrl_SIf_PBC
TYPE T_Ctrl_SIf_PBC :
STRUCT
	///configuration
	Cfg: T_Ctrl_SIf_PBC_Cfg;
	///parameter
	Par: T_Ctrl_SIf_PBC_Par;
	///current values
	Cur: T_Ctrl_SIf_PBC_Cur;
	///io input
	In: T_Ctrl_SIf_PBC_In;
	///io output
	Out: T_Ctrl_SIf_PBC_Out;
	///alarm number used in this controller
	Alm: ARRAY[1..E_ALM_PBC.MAX_E_ALM_PBC] OF T_Ctrl_Alm;
	///interlock of output/movements
	Ilk: T_Ctrl_SIf_PBC_Ilk;
END_STRUCT
END_TYPE

// POUs/Controller/Lvl2/PBC [Paper Buffer Controller]/T_Ctrl_SIf_PBC_Cfg
TYPE T_Ctrl_SIf_PBC_Cfg :
STRUCT
	/// True : Use the turn table sensor to detect ejects.
	bolUseTurnTableSensorForEject: BOOL;
	/// Enable the Data Channel to Saber to send the read barcodes to Saber
	bolEnableDataChannel: BOOL;
	/// Airpressure unit for the granulate available
	bolGranulatAirPressureUnitAvailable: BOOL;
	/// Enable or Disable the Saber Stop DeStack to do manual operation
	bolEnableSaberStopDeStack: BOOL;
END_STRUCT
END_TYPE

// POUs/Controller/Lvl2/PBC [Paper Buffer Controller]/T_Ctrl_SIf_PBC_Cur
TYPE T_Ctrl_SIf_PBC_Cur :
STRUCT
	/// How many papers are in the buffer. -1 = Paper count unknown
	intPaperInBufferCount: INT;
	/// Last Paper to eject count parameter
	uinPaperToEjectParameter: UINT;
	/// Actual count of the paper ejected 
	uinPaperToEjectCount: UINT;
	/// [ms] Time from sheet to sheet ejection in multi eject mode.
	uinSheetToSheetTime: UINT;
	/// Was paper before Eject available
	bolPaperBeforeEjectAvailable: BOOL;
	/// Paper to paper Timeout
	uinPaperToPaperTime_ms: UINT;
	/// Last Read Barcode			
	udiLastBarcode: UDINT;
	/// Total Paper Counter / Also used to signal a new Barcode read.			
	udiBarcodeChanged: UDINT;
END_STRUCT
END_TYPE

// POUs/Controller/Lvl2/PBC [Paper Buffer Controller]/T_Ctrl_SIf_PBC_Ilk
TYPE T_Ctrl_SIf_PBC_Ilk :
STRUCT
END_STRUCT
END_TYPE

// POUs/Controller/Lvl2/PBC [Paper Buffer Controller]/T_Ctrl_SIf_PBC_In
TYPE T_Ctrl_SIf_PBC_In :
STRUCT
	/// This sensor shows if the buffer reaches his capacity limits
	bolPaperAvailableExit: BASE_PLC.T_Ctrl_IoBool;
	/// Shows if there is paper available in the buffer
	bolPaperAvailableEntry: BASE_PLC.T_Ctrl_IoBool;
	/// Shows if there is a paper on the output of the buffer
	bolCapacityReached: BASE_PLC.T_Ctrl_IoBool;
	/// Double paper detection
	bolDoublePaperDetection: BASE_PLC.T_Ctrl_IoBool;
	/// Turn Table Mid Sensor
	bolTurnTableMiddleSensor: BASE_PLC.T_Ctrl_IoBool;
	/// Airpressure Ok
	bolAirPressorOk: BASE_PLC.T_Ctrl_IoBool;
END_STRUCT
END_TYPE

// POUs/Controller/Lvl2/PBC [Paper Buffer Controller]/T_Ctrl_SIf_PBC_Out
TYPE T_Ctrl_SIf_PBC_Out :
STRUCT
	/// Air on the Airpressure supply unit on:
	bolAirOn: BASE_PLC.T_Ctrl_IoBool;
END_STRUCT
END_TYPE

// POUs/Controller/Lvl2/PBC [Paper Buffer Controller]/T_Ctrl_SIf_PBC_Par
TYPE T_Ctrl_SIf_PBC_Par :
STRUCT
	/// [ms] Paper transport timeout - Time that paper is allowed to have for the transport to the front.
	udiPaperTransportTime: UDINT;
	/// Sheet to output with one run command.  0 = endless until stop
	udiSheetToEject: UDINT;
	/// [ms] Time from sheet to sheet ejection in multi eject mode in Auto Mode.
	udiSheetToSheetTime: UDINT;
	/// [ms] Time from sheet to sheet ejection in multi eject mode in Manual Mode.
	udiManualSheetToSheetTime_ms: UDINT;
	/// [ms] Paper transport time simulation
	udiSimPaperTransportTime: UDINT;
	/// [ms] Paper to paper transport time simulation
	udiSimPaperToPaperTransportTime: UDINT;
	/// # of retries for paper transport. 
	udiPaperInjectRetries: UDINT;
	/// Enable Double Paper detection
	bolEnableDoublePaperDetection: BOOL;
	/// [ms] Double Paper detection sensor debounce time
	udiDoublePaperDebounceTime_ms: UDINT;
	/// [ms] Retry Pause Time
	udiPaperInjectRetryPauseTime_ms: UDINT;
	/// Automatic or Manual DeStacking Mode
	bolAutomaticMode: BOOL;
	/// Indicates that the controller must not release any item but can still collect new items (RUN state). This flag is normally set by LineControl.
	bolStopReleaseItems: BOOL;
END_STRUCT
END_TYPE

// POUs/Controller/Lvl2/PCE [Paper Belt Corner Element]/helper/T_PCE
TYPE T_PCE :
STRUCT
	io:		T_PCE_IO;
	ctrl:	T_PCE_CTRL;
	id:		T_PCE_ID;
END_STRUCT
END_TYPE

// POUs/Controller/Lvl2/PCE [Paper Belt Corner Element]/helper/T_PCE_CTRL
TYPE T_PCE_CTRL :
STRUCT
	fbPce: FB_PCE;
	fbPce_PtbIn: FB_PTB;
	fbPce_PtbIn_Umc: FB_UMC;
	fbPce_PtbIn_Vpc: FB_VPC;
	fbPce_PtbOut: FB_PTB;
	fbPce_PtbOut_Umc: FB_UMC;
END_STRUCT
END_TYPE

// POUs/Controller/Lvl2/PCE [Paper Belt Corner Element]/helper/T_PCE_ID
TYPE T_PCE_ID :
STRUCT
	Pce: INT;
	Pce_PtbIn: INT;
	Pce_PtbIn_Umc: INT;
	Pce_PtbIn_Vpc: INT;
	Pce_PtbOut: INT;
	Pce_PtbOut_Umc: INT;
END_STRUCT
END_TYPE

// POUs/Controller/Lvl2/PCE [Paper Belt Corner Element]/helper/T_PCE_IO
TYPE T_PCE_IO :
STRUCT
	In_bolInputSensor: REFERENCE TO BOOL;
	In_bolOutputSensor: REFERENCE TO BOOL;
	In_bolCornerSensor: REFERENCE TO BOOL;
	Out_bolVacuumValveIn: REFERENCE TO BOOL;
	Out_bolVacuumValveOut: REFERENCE TO BOOL;

	In_uinUmcIn_Status: REFERENCE TO UINT;
	In_uinUmcIn_ActualSpeed: REFERENCE TO UINT;
	In_uinUmcIn_SetSpeed: REFERENCE TO UINT;
	In_uinUmcIn_IOData1: REFERENCE TO WORD;
	In_uinUmcIn_ECatState: REFERENCE TO UINT;
	In_strUmcIn_ECatNetId: REFERENCE TO AMSNETID;
	In_uinUmcIn_ECatPort: REFERENCE TO WORD;
	Out_uinUmcIn_Control: REFERENCE TO UINT;
	Out_uinUmcIn_SetSpeed: REFERENCE TO UINT;
	
	In_uinUmcOut_Status: REFERENCE TO UINT;
	In_uinUmcOut_ActualSpeed: REFERENCE TO UINT;
	In_uinUmcOut_SetSpeed: REFERENCE TO UINT;
	In_uinUmcOut_IOData1: REFERENCE TO WORD;
	In_uinUmcOut_ECatState: REFERENCE TO UINT;
	In_strUmcOut_ECatNetId: REFERENCE TO AMSNETID;
	In_uinUmcOut_ECatPort: REFERENCE TO WORD;
	Out_uinUmcOut_Control: REFERENCE TO UINT;
	Out_uinUmcOut_SetSpeed: REFERENCE TO UINT;
	
	In_bolVpc_VacuumSensor: REFERENCE TO BOOL;
	In_bolVpc_PumpOk: REFERENCE TO BOOL;
	Out_bolVpc_PumpOn: REFERENCE TO BOOL;
END_STRUCT
END_TYPE

// POUs/Controller/Lvl2/PCE [Paper Belt Corner Element]/E_ALM_PCE
TYPE E_ALM_PCE :
(
	PaperSensorError := 1,
	MAX_E_ALM_PCE
);
END_TYPE

// POUs/Controller/Lvl2/PCE [Paper Belt Corner Element]/T_Ctrl_SIf_PCE
TYPE T_Ctrl_SIf_PCE :
STRUCT
	///configuration
	Cfg: T_Ctrl_SIf_PCE_Cfg;
	///parameter
	Par: T_Ctrl_SIf_PCE_Par;
	///current values
	Cur: T_Ctrl_SIf_PCE_Cur;
	///io input
	In: T_Ctrl_SIf_PCE_In;
	///io output
	Out: T_Ctrl_SIf_PCE_Out;
	///alarm number used in this controller
	Alm: ARRAY[1..MAX_E_ALM_PCE] OF T_Ctrl_Alm;
	///interlock of output/movements
	Ilk: T_Ctrl_SIf_PCE_Ilk;
END_STRUCT
END_TYPE

// POUs/Controller/Lvl2/PCE [Paper Belt Corner Element]/T_Ctrl_SIf_PCE_Cfg
TYPE T_Ctrl_SIf_PCE_Cfg :
STRUCT
END_STRUCT
END_TYPE

// POUs/Controller/Lvl2/PCE [Paper Belt Corner Element]/T_Ctrl_SIf_PCE_Cur
TYPE T_Ctrl_SIf_PCE_Cur :
STRUCT
	/// [mm/s] Belt speed
	uinBeltSpeed: UINT;
END_STRUCT
END_TYPE

// POUs/Controller/Lvl2/PCE [Paper Belt Corner Element]/T_Ctrl_SIf_PCE_Ilk
TYPE T_Ctrl_SIf_PCE_Ilk :
STRUCT
END_STRUCT
END_TYPE

// POUs/Controller/Lvl2/PCE [Paper Belt Corner Element]/T_Ctrl_SIf_PCE_In
TYPE T_Ctrl_SIf_PCE_In :
STRUCT
	/// 0 = Paper not here; 1 = Paper detected
	bolPaperAvailable: BASE_PLC.T_Ctrl_IoBool;
END_STRUCT
END_TYPE

// POUs/Controller/Lvl2/PCE [Paper Belt Corner Element]/T_Ctrl_SIf_PCE_Out
TYPE T_Ctrl_SIf_PCE_Out :
STRUCT
	/// Paper Incoming Belt - 0 = Vacuum Valve Closed;  1 = Vacuum valve open
	bolVacuumValveIn: BASE_PLC.T_Ctrl_IoBool;
	/// Paper Outgoing Belt - 0 = Vacuum Valve Closed;  1 = Vacuum valve open
	bolVacuumValveOut: BASE_PLC.T_Ctrl_IoBool;
END_STRUCT
END_TYPE

// POUs/Controller/Lvl2/PCE [Paper Belt Corner Element]/T_Ctrl_SIf_PCE_Par
TYPE T_Ctrl_SIf_PCE_Par :
STRUCT
	/// [ms] Paper entry delay time. Time delay between detection and switching the vacuum
	uinPaperEntryDelayTime_ms: UDINT;
	/// [ms] Paper exit time
	uinPaperExitTime_ms: UDINT;
	/// [ms] Simulation Paper exit time
	uinSimPaperExitTime_ms: UDINT;
END_STRUCT
END_TYPE

// POUs/Controller/Lvl2/PST [Paper Stacker]/helper/T_PST
TYPE T_PST :
STRUCT
	io:		T_PST_IO;
	ctrl:	T_PST_CTRL;
	id:		T_PST_ID;
END_STRUCT
END_TYPE

// POUs/Controller/Lvl2/PST [Paper Stacker]/helper/T_PST_CTRL
TYPE T_PST_CTRL :
STRUCT
	fbPst: FB_PST;
	fbPst_Ptb: FB_PTB;
	fbPst_Ptb_Umc: FB_UMC;
	fbPst_Ptb_Vpc: FB_VPC;
END_STRUCT
END_TYPE

// POUs/Controller/Lvl2/PST [Paper Stacker]/helper/T_PST_ID
TYPE T_PST_ID :
STRUCT
	Pst: INT;
	Pst_Ptb: INT;
	Pst_Ptb_Umc: INT;
	Pst_Ptb_Vpc: INT;
END_STRUCT
END_TYPE

// POUs/Controller/Lvl2/PST [Paper Stacker]/helper/T_PST_IO
TYPE T_PST_IO :
STRUCT
	In_bolSensorPaperAtOperatorPos: REFERENCE TO BOOL;
	In_bolSensorStopperPosition: REFERENCE TO BOOL;
	In_bolSensorInfeed: REFERENCE TO BOOL;
	In_bolSensorOutfeed: REFERENCE TO BOOL;
	
	In_bolPtb_InputSensor: REFERENCE TO BOOL;
	In_bolPtb_OutputSensor: REFERENCE TO BOOL;
	
	In_bolPtb_Vpc_VacuumSensor: REFERENCE TO BOOL;
	In_bolPtb_Vpc_PumpOk: REFERENCE TO BOOL;
	Out_bolPtb_Vpc_PumpOn: REFERENCE TO BOOL;
	
	In_uinPtb_Umc_Status: REFERENCE TO UINT;
	In_uinPtb_Umc_ActualSpeed: REFERENCE TO UINT;
	In_uinPtb_Umc_SetSpeed: REFERENCE TO UINT;
	In_uinPtb_Umc_IOData1: REFERENCE TO WORD;
	In_uinPtb_Umc_ECatState: REFERENCE TO UINT;
	In_strPtb_Umc_ECatNetId: REFERENCE TO AMSNETID;
	In_uinPtb_Umc_ECatPort: REFERENCE TO WORD;
	Out_uinPtb_Umc_Control: REFERENCE TO UINT;
	Out_uinPtb_Umc_SetSpeed: REFERENCE TO UINT;
END_STRUCT
END_TYPE

// POUs/Controller/Lvl2/PST [Paper Stacker]/E_ALM_PST
TYPE E_ALM_PST :
(
	StackIncomplete := 1,
	NeedsEjectCommand := 2,
	StackOkButLastCodeNotRight := 3,
	StackNotOkButLastCodeRight := 4,
	ReadingBarcodeFailedAfterXRetries := 5,
	NewPaperDetectedDuringEjecting := 6,
	NewPaperDetectedWhileBarcodeReading := 7,
	MAX_E_ALM_PST
);
END_TYPE

// POUs/Controller/Lvl2/PST [Paper Stacker]/T_Ctrl_SIf_PST
TYPE T_Ctrl_SIf_PST :
STRUCT
	///configuration
	Cfg: T_Ctrl_SIf_PST_Cfg;
	///parameter
	Par: T_Ctrl_SIf_PST_Par;
	///current values
	Cur: T_Ctrl_SIf_PST_Cur;
	///io input
	In: T_Ctrl_SIf_PST_In;
	///alarm number used in this controller
	Alm: ARRAY[1..E_ALM_PST.MAX_E_ALM_PST] OF T_Ctrl_Alm;
END_STRUCT
END_TYPE

// POUs/Controller/Lvl2/PST [Paper Stacker]/T_Ctrl_SIf_PST_Cfg
TYPE T_Ctrl_SIf_PST_Cfg :
STRUCT
	/// Enable data channel to saber
	bolEnableDataChannel	: BOOL;
	/// Number of retry barcode read command if failed
	uinNumOfRetryRead		: UINT;
	/// Rotation direction for ejecting
	/// LEFT  = 1
	/// RIGHT = 2
	usiEjectingDirection	: INT;
	/// Rotation direction for reverse
	/// LEFT  = 1
	/// RIGHT = 2
	usiReverseDirection		: INT;
	/// Enable PST controlled Eject
	bolEnablePstEjectControl: BOOL;
END_STRUCT
END_TYPE

// POUs/Controller/Lvl2/PST [Paper Stacker]/T_Ctrl_SIf_PST_Cur
TYPE T_Ctrl_SIf_PST_Cur :
STRUCT
	/// # of papers in the stack
	uinStackHight: UINT;
	/// Total number of stacks ejected 
	udiNumOfStacksEjectedTotal: UDINT;
	/// Indicates that the last stacking job was incomplete. Run command not possible. Needs eject command from saber.
	bolStackIncomplete: BOOL;
END_STRUCT
END_TYPE

// POUs/Controller/Lvl2/PST [Paper Stacker]/T_Ctrl_SIf_PST_In
TYPE T_Ctrl_SIf_PST_In :
STRUCT
	/// Sensor detects if a paper is at the operator position
	bolSensorPaperAtOperatorPos: BASE_PLC.T_Ctrl_IoBoolDebounced;
	/// Sensor detects the stopper position (TRUE = stopper position down , FALSE = stopper position up)
	bolSensorStopperPosition: BASE_PLC.T_Ctrl_IoBoolDebounced;
	/// Sensor detects paper on outfeed position 
	bolSensorOutfeed: BASE_PLC.T_Ctrl_IoBoolDebounced;
	/// Sensor detects paper on infeed position
	bolSensorInfeed: BASE_PLC.T_Ctrl_IoBool;
END_STRUCT
END_TYPE

// POUs/Controller/Lvl2/PST [Paper Stacker]/T_Ctrl_SIf_PST_Par
TYPE T_Ctrl_SIf_PST_Par :
STRUCT
	/// Stack hight in # of paper to eject. Sent by saber. 
	uinStackHight: UINT;
	/// Last barcode in stack. Sent by saber. 
	/// If stack hight is reached and last barcode in stack detected, stacker automatically eject the whole stack.
	uliLastBarCodeInStack: ULINT;
	/// [mm/s] Belt reverse speed to bring stopper back to up position
	uinBeltReverseSpeed_mmsec: UINT;
	/// [mm/s] Belt speed for ejecting the whole stack
	uinBeltEjectSpeed_mmsec: UINT;
	/// [ms] Paper is at operator position delay time
	udiPaperAtOpPosDebounceTime_ms: UDINT;
	/// [ms] Stopper position delay time
	udiStopperPosDebounceTime_ms: UDINT;
	/// [ms] Outfeed sensor delay time
	udiSensorOutfeedDebounceTime_ms: UDINT;
	/// [ms] Stack eject delay time - Delay before belt starts to eject the stack if hight is reached.
	udiStackEjectDelayTime_ms: UDINT;
	/// [ms] Stack ejecting time - Time for how long the belt should move in eject direction 
	udiStackEjectingTime_ms: UDINT;
	/// [ms] Belt reverse delay time - Delay before belt starts moving backward after ejecting stack.
	udiBeltReverseDelayTime_ms: UDINT;
	/// [ms] Barcode reader trigger delay time - Delay time, until a read command will be executed, after a new paper was detected at infeed sensor.
	udiBarcodeReaderTriggerDelayTime_ms: UDINT;
	/// [ms] Simulation time paper infeed stroke
	udiSimTimePaperInfeedStroke_ms: UDINT;
END_STRUCT
END_TYPE

// POUs/Controller/Lvl2/PST [Paper Stacker]/T_ItemPaperInfo
{attribute 'enable_dynamic_creation' := ''}
TYPE T_ItemPaperInfo :
STRUCT
	/// Position in the stack
	uinPosInStack: UINT;
	/// Barcode of the paper
	uliBarCode: ULINT;
END_STRUCT
END_TYPE

// POUs/Controller/Lvl2/PTS [Paper Turning Station]/helper/T_PTS
TYPE T_PTS :
STRUCT
	io			: T_PTS_IO;
	ctrl		: T_PTS_CTRL;
	id			: T_PTS_ID;
END_STRUCT
END_TYPE

// POUs/Controller/Lvl2/PTS [Paper Turning Station]/helper/T_PTS_CTRL
TYPE T_PTS_CTRL :
STRUCT
	fbPts_RAX_POD		: FB_POD;
	fbPts_RAX			: FB_RAX;
	fbPts_Ptb			: FB_PTB;
	fbPts_Ptb_Umc		: FB_UMC;
	fbPts_Ptb_Vpc		: FB_VPC;
	fbPts_Mdc_Umc		: FB_UMC;
	fbPts_Mdc			: FB_MDC;
	fbPts				: FB_PTS;
END_STRUCT
END_TYPE

// POUs/Controller/Lvl2/PTS [Paper Turning Station]/helper/T_PTS_ID
TYPE T_PTS_ID :
STRUCT
	Pts				: INT;
	Pts_Ptb			: INT;
	Pts_Ptb_Umc		: INT;
	Pts_Ptb_Vpc		: INT;
	Pts_Mdc			: INT;
	Pts_Mdc_Umc		: INT;
	/// New Servo Drive PLC opend driver
	Pts_RAX_POD		: INT;
	/// New Servo Drive
	Pts_RAX			: INT;
END_STRUCT
END_TYPE

// POUs/Controller/Lvl2/PTS [Paper Turning Station]/helper/T_PTS_IO
TYPE T_PTS_IO :
STRUCT
	In_bolPaperSensor: REFERENCE TO BOOL;
	
	In_bolMdc_CrossPositionSensor: REFERENCE TO BOOL;
	In_bolMdc_TablePositionSensor: REFERENCE TO BOOL;
	
	In_uinMdc_Umc_Status: REFERENCE TO UINT;
	In_uinMdc_Umc_ActualSpeed: REFERENCE TO UINT;
	In_uinMdc_Umc_SetSpeed: REFERENCE TO UINT;
	In_uinMdc_Umc_IOData1: REFERENCE TO WORD;
	In_uinMdc_Umc_ECatState: REFERENCE TO UINT;
	In_strMdc_Umc_ECatNetId: REFERENCE TO AMSNETID;
	In_uinMdc_Umc_ECatPort: REFERENCE TO WORD;
	Out_uinMdc_Umc_Control: REFERENCE TO UINT;
	Out_uinMdc_Umc_SetSpeed: REFERENCE TO UINT;
	
	In_uinPtb_Umc_Status: REFERENCE TO UINT;
	In_uinPtb_Umc_ActualSpeed: REFERENCE TO UINT;
	In_uinPtb_Umc_SetSpeed: REFERENCE TO UINT;
	In_uinPtb_Umc_IOData1: REFERENCE TO WORD;
	In_uinPtb_Umc_ECatState: REFERENCE TO UINT;
	In_strPtb_Umc_ECatNetId: REFERENCE TO AMSNETID;
	In_uinPtb_Umc_ECatPort: REFERENCE TO WORD;
	Out_uinPtb_Umc_Control: REFERENCE TO UINT;
	Out_uinPtb_Umc_SetSpeed: REFERENCE TO UINT;
	
	In_bolPtb_Vpc_VacuumSensor: REFERENCE TO BOOL;
	In_bolPtb_Vpc_PumpOk: REFERENCE TO BOOL;
	Out_bolPtb_Vpc_PumpOn: REFERENCE TO BOOL;
	
	In_bolRax_PositionSensor: REFERENCE TO BOOL;
	//TODO
END_STRUCT
END_TYPE

// POUs/Controller/Lvl2/PTS [Paper Turning Station]/E_ALM_PTS
TYPE E_ALM_PTS :
(
	PaperTransport 				:= 1,
	ModeParameter 				:= 2,
	TurnTableConfigMissmatch	:= 3,
	MAX_E_ALM_PTS
);
END_TYPE

// POUs/Controller/Lvl2/PTS [Paper Turning Station]/E_PTS_MODE
TYPE E_PTS_MODE :
(
	Automatic := -2,
	Distribute := -1,
	FixA := 0,
	FixB := 1,
	FixC := 2,
	MAX_E_PTS_MODE
);
END_TYPE

// POUs/Controller/Lvl2/PTS [Paper Turning Station]/T_Ctrl_SIf_PTS
TYPE T_Ctrl_SIf_PTS :
STRUCT
	///configuration
	Cfg: T_Ctrl_SIf_PTS_Cfg;
	///parameter
	Par: T_Ctrl_SIf_PTS_Par;
	///current values
	Cur: T_Ctrl_SIf_PTS_Cur;
	///io input
	In: T_Ctrl_SIf_PTS_In;
	///io output
	Out: T_Ctrl_SIf_PTS_Out;
	///alarm number used in this controller
	Alm: ARRAY[1..MAX_E_ALM_PTS] OF T_Ctrl_Alm;
	///interlock of output/movements
	Ilk: T_Ctrl_SIf_PTS_Ilk;
END_STRUCT
END_TYPE

// POUs/Controller/Lvl2/PTS [Paper Turning Station]/T_Ctrl_SIf_PTS_Cfg
TYPE T_Ctrl_SIf_PTS_Cfg :
STRUCT
	/// Turns the barcode reader intelligence on. This makes the PTS nearly self sustained. 
	bolBarcodeReaderAvailable: BOOL;
	/// If there is no barcode but a sensor at the end of the entry belt 
	bolEntrySensorAvailable: BOOL;
	/// Paper Input and Ouput Positions for the fixed modes
	aFixPosDef: ARRAY[0..(E_PTS_MODE.MAX_E_PTS_MODE - 1)] OF T_PTS_InOutPositions;
	/// Automatic Mode Input and Output Positions
	aAutoPosDef: ARRAY[0..(cPTS_MAX_AUTOPOS - 1)] OF T_PTS_InOutPositions;
	/// Automatic Mode Default Input Positions
	aDefaultAutoPos: UINT;
	/// Paper Input and Ouput Positions for the fixed modes
	aDistributionPositionDefinition: ARRAY[0..(PTS_CmdState.cPTS_MAX_DISTRIBUTION - 1)] OF E_PTS_MODE;
	/// Start positioning the malteser wheel before turning
	bolPositionMalteserEnable: BOOL;
	/// Use Servo Axis instead of Malteser for turning
	bolRaxEnable: BOOL;
END_STRUCT
END_TYPE

// POUs/Controller/Lvl2/PTS [Paper Turning Station]/T_Ctrl_SIf_PTS_Cur
TYPE T_Ctrl_SIf_PTS_Cur :
STRUCT
	/// Actual Sheet In- Out- Positions
	rInOutPosition: T_PTS_InOutPositions;
	/// Saves the last executed distribution index
	iActualDistributionIndex: INT;
	/// [ms] Time to wait after paper was detected before to turn.
	udiPaperInTurnDelayTime: UDINT;
	/// [ms] Time to wait after paper is not detected anymore before to turn back.
	udiPaperOutTurnDelayTime: UDINT;
	// Count of turn movements in long term test
	udiPTS_Counter: UDINT;
END_STRUCT
END_TYPE

// POUs/Controller/Lvl2/PTS [Paper Turning Station]/T_Ctrl_SIf_PTS_Ilk
TYPE T_Ctrl_SIf_PTS_Ilk :
STRUCT
END_STRUCT
END_TYPE

// POUs/Controller/Lvl2/PTS [Paper Turning Station]/T_Ctrl_SIf_PTS_In
TYPE T_Ctrl_SIf_PTS_In :
STRUCT
	/// This sensor shows if the paper is at the middle table possition
	bolPaperAvailable: BASE_PLC.T_Ctrl_IoBool;
	/// This sensor shows if the paper is available at the exit of the input belt
	bolPaperAtBeltExit: BASE_PLC.T_Ctrl_IoBool;
END_STRUCT
END_TYPE

// POUs/Controller/Lvl2/PTS [Paper Turning Station]/T_Ctrl_SIf_PTS_Out
TYPE T_Ctrl_SIf_PTS_Out :
STRUCT
END_STRUCT
END_TYPE

// POUs/Controller/Lvl2/PTS [Paper Turning Station]/T_Ctrl_SIf_PTS_Par
TYPE T_Ctrl_SIf_PTS_Par :
STRUCT
	/// [ms] Time to wait after paper was detected before to turn.
	udiPaperInTurnDelayTime: UDINT;
	/// [ms] Time to wait after paper is not detected anymore before to turn back.
	udiPaperOutTurnDelayTime: UDINT;
	/// [ms] Timeout for the time the Paper can have between Barcode reader and Paper on table sensor.
	udiPaperBarcodeToInputSensorTime: UDINT;
	/// Mode for turning
	eMode: E_PTS_MODE;
	/// [ms] Simulation Timeout for the time the Paper can have between Barcode reader and Paper on table sensor.
	udiSimPaperBarcodeToInputSensorTime: UDINT;
	// Activate long time test
	bolLongTimeTestEnable: BOOL;
END_STRUCT
END_TYPE

// POUs/Controller/Lvl2/PTS [Paper Turning Station]/T_PTS_InOutPositions
TYPE T_PTS_InOutPositions :
STRUCT
	uinInput: UINT;
	uinOutput: UINT;
	eDirection: E_TURN_DIRECTION;
END_STRUCT
END_TYPE

// POUs/Controller/Utility/Data Channel/OvenMessage/T_Oven_DCH
{attribute 'enable_dynamic_creation' := ''}
TYPE T_Oven_DCH :
STRUCT
	rBaseInfo: T_ItemBase;
	/// Paper ID
	udiIdentification: ULINT;
	/// Recipe  process parameter
	/// --------------------------------------------------------------
	/// Oven Data
	bTrash: BOOL;
	diTimeInOven_s: DINT;
	diTemperature_mc: ARRAY[0..(MAX_NUMBER_OF_OVEN_MODULES - 1)] OF DINT;
	diAirflow_prc: ARRAY[0..(MAX_NUMBER_OF_OVEN_MODULES - 1)] OF DINT;
END_STRUCT
END_TYPE

// POUs/Controller/Utility/Data Channel/OvenMessage/T_OvenSendData
TYPE T_OvenSendData :
STRUCT
	fbDataChannel: FB_IdBaseSendDch;
	rDataChannelItem: T_Oven_DCH;
	fbFifo: FB_DataChannelSenderFifo;
END_STRUCT
END_TYPE

// GVLs/Constants
VAR_GLOBAL CONSTANT
	
	// Oven
	// ----------------------------------------------------------------------
	MAX_INT: INT := 32767;
	MIN_INT: INT := -32768;
	MAX_NUMBER_OF_OVEN_MODULES: UINT := 8;
	WRITE_BUFFER_LENGTH: UDINT := 98;
	READ_BUFFER_LENGTH: UDINT := 103;
	
END_VAR

// POUs/Controller/Driver/IBH (IBH Link)/IBH_CmdState
VAR_GLOBAL CONSTANT
	///ctrl commands definitions
	///specific commands >200 - every command has to be a even number
	cCMD_CONNECT: INT := 202;
	cCMD_WRITE: INT := 204;
	cCMD_READ: INT := 206;
	cCMD_DISCONNECT: INT := 208;
	///ctrl specific states definitions
	cSTA_CONNECTBusy: INT := 201;
	cSTA_CONNECT: INT := 202;
	cSTA_WRITEBusy: INT := 203;
	cSTA_WRITE: INT := 204;
	cSTA_READBusy: INT := 205;
	cSTA_READ: INT := 206;
	cSTA_DISCONNECTBusy: INT := 207;
	cSTA_DISCONNECT: INT := 208;
	cSTA_SUB_1: INT := 301;
	cSTA_SUB_2: INT := 302;
	cSTA_SUB_3: INT := 303;
	cSTA_SUB_4: INT := 304;
	cSTA_SUB_5: INT := 305;
END_VAR

// POUs/Controller/Driver/POD (PLCopen Driver)/POD_Cmd
VAR_GLOBAL CONSTANT
	/// Switch controller on 
	cPOD_STA_PowerOff: INT := 0;
	/// Error
	cPOD_STA_Error: INT := 256;
	cPOD_STA_WaitForJob: INT := 1000;
	cPOD_STA_PowerOnBusy: INT := 1001;
	/// Homing 
	cPOD_STA_HomeBusy: INT := 1006;
	/// Start move with relative move distance 
	cPOD_STA_RelMoveBusy: INT := 1007;
	/// Start move with absolute target position 
	cPOD_STA_AbsMoveBusy: INT := 1010;
	/// Start move in positive direction 
	cPOD_STA_PosMoveBusy: INT := 1011;
	cPOD_STA_PosMove: INT := 1012;
	/// Start move in negative direction 
	cPOD_STA_NegMoveBusy: INT := 1013;
	cPOD_STA_NegMove: INT := 1014;
	/// controller on standstill
	cPOD_STA_StopBusy: INT := 1015;
	/// controller on standstill
	cPOD_STA_QStopBusy: INT := 1017;
	/// controller on standstill
	cPOD_STA_NegJogBusy: INT := 1019;
	/// controller on standstil	
	cPOD_STA_PosJogBusy: INT := 1021;
	cPOD_STA_ModMoveBusy: INT := 1023;
	cPOD_STA_ModMove: INT := 1024;
	cPOD_STA_StorePara: INT := 1050;
	cPOD_STA_WritePara: INT := 1052;
	/// ctrl commands definitions
	/// specific commands >200 - every command has to be a even number
	cPOD_CMD_DONE: INT := -1;
	/// Switch controller on 
	cPOD_CMD_CTRL_ON: INT := 1002;
	/// Switch controller off 
	cPOD_CMD_CTRL_OFF: INT := 1004;
	/// Homing 
	cPOD_CMD_HOME: INT := 1006;
	/// Start move with relative move distance 
	cPOD_CMD_REL_MOVE: INT := 1008;
	/// Start move with absolute target position 
	cPOD_CMD_ABS_MOVE: INT := 1010;
	/// Start move in positive direction 
	cPOD_CMD_POS_MOVE: INT := 1012;
	/// Start move in negative direction 
	cPOD_CMD_NEG_MOVE: INT := 1014;
	/// Stop movement with controller on 
	cPOD_CMD_STOP: INT := 1016;
	/// Emergency stop with controller off 
	cPOD_CMD_EMCY_STOP_CTRL_OFF: INT := 1018;
	/// Start move in positive direction 
	cPOD_CMD_POS_JOG: INT := 1020;
	cPOD_CMD_NEG_JOG: INT := 1022;
	/// Start move with modulo positionining (based on modulofactor defined in axis parameter!)
	cPOD_CMD_MOD_MOVE: INT := 1024;
	cPOD_CMD_STORE_PARAMETER: INT := 1050;
	cPOD_CMD_WRITE_PARAMETER: INT := 1052;
	/// Service Jobs (parallel to active job)
	cPOD_SCMD_WRITE_PARA: INT := 2002;
	cPOD_SCMD_READ_PARA: INT := 2004;
	cPOD_SCMD_RESET_ABSENCODER: INT := 2006;
	cPOD_SCMD_WRITE_PARA_NC: INT := 2008;
	cPOD_SCMD_READ_PARA_NC: INT := 2010;
END_VAR

// POUs/Controller/Driver/POD (PLCopen Driver)/POD_Const
VAR_GLOBAL
END_VAR

// POUs/Controller/Driver/TCP (TCP communication driver)/TCP_CmdState
VAR_GLOBAL CONSTANT
	/// ctrl commands definitions
	/// specific commands >200 - every command has to be a even number
	cCMD_Close: INT := 202;
	cCMD_Connect: INT := 204;
	/// ctrl specific states definitions
	cSTA_CloseBusy: INT := 201;
	cSTA_Close: INT := 202;
	cSTA_ConnectBusy: INT := 203;
	cSTA_Connect: INT := 204;
END_VAR

// POUs/Controller/Driver/TCP (TCP communication driver)/TCP_Constants
VAR_GLOBAL CONSTANT
	/// Define length of data buffer. Max. 900 Byte
	MAX_DATASET_SIZE: UDINT := 900;
END_VAR

// POUs/Controller/Lvl0/JCL (Jetter Client)/JCL_CmdState
VAR_GLOBAL CONSTANT
	/// Preparing jetter for production
	cCMD_Standby: INT := 202;
	/// Start calibration routine for MM camera system
	cCMD_Calibration: INT := 204;
	/// Start automatic cleaning cycle for both printheads
	cCMD_CleanPrintHeads: INT := 206;
	/// Reset pending alarms
	cCMD_ResetAlarm: INT := 230;
	/// Send back the state msg.
	cCMD_RequestState: INT := 240;
	/// ctrl specific states definitions
	cSTA_StandbyBusy: INT := 201;
	cSTA_Standby: INT := cCMD_Standby;
	cSTA_ConnectBusy: INT := 250;
	cSTA_CleanPrintHeadsBusy: INT := 205;
	cSTA_CleanPrintHeads: INT := cCMD_CleanPrintHeads;
	cSTA_CalibrationBusy: INT := 203;
	cSTA_Calibration: INT := cCMD_Calibration;
	cSTA_ParkBusy: INT := 211;
	cSTA_MaintenanceBusy: INT := 208;
	cSTA_MaintenanceInWork: INT := 209;
	cSTA_MaintenanceDone: INT := 210;
	cSTA_MANUALMODE: INT := 212;
	/// sub states
	cSUB_WaitingForConnection: INT := 300;
	cSUB_WaitingForState: INT := 301;
	cSUB_WaitingSocketClosed: INT := 302;
	cSUB_SendPon: INT := 303;
	cSUB_Done: INT := 999;
END_VAR

// POUs/Controller/Lvl0/JCL (Jetter Client)/JCL_Constants
VAR_GLOBAL CONSTANT
	/// MsgID (valid for jetter TCP server protocol)
	JCL_MsgId_Command: UINT := 1;
	JCL_MsgId_State: UINT := 2;
	JCL_MsgId_Alarm: UINT := 4;
	JCL_MsgId_PrintDone: UINT := 5;
	JCL_MsgId_ReqCleaning: UINT := 6;
	/// Jetter CMD (valid for jetter TCP server protocol)	
	JCL_CMD_PowerOn: USINT := 2;
	JCL_CMD_Off: USINT := 6;
	JCL_STA_Standby: USINT := 202;
	JCL_CMD_Standby: USINT := 202;
	JCL_CMD_Run: USINT := 10;
	JCL_CMD_CleanPrintHeads: USINT := 206;
	JCL_CMD_Calibration: USINT := 204;
	JCL_CMD_ResetAlarm: USINT := 230;
	JCL_CMD_RequestState: USINT := 240;
END_VAR

// POUs/Controller/Lvl0/RAX(Rotative Axis)/RAX_CmdState
VAR_GLOBAL CONSTANT
	///ctrl commands definitions
	///specific commands >200 - every command has to be a even number
	cCMD_HOME: INT := 202;
	cCMD_POS: INT := 204;
	cCMD_JOG_NEG: INT := 210;
	cCMD_JOG_POS: INT := 212;
	cCMD_REL_POS: INT := 214;
	cCMD_TURN: INT := 216;
	///ctrl specific states definitions
	cSTA_POSBusy: INT := 203;
	cSTA_POS: INT := RAX_CmdState.cCMD_POS;
	cSTA_REL_POSBusy: INT := 213;
	cSTA_REL_POS: INT := RAX_CmdState.cCMD_REL_POS;
	cSTA_JOG_NEG: INT := RAX_CmdState.cCMD_JOG_NEG;
	cSTA_JOG_POS: INT := RAX_CmdState.cCMD_JOG_POS;
	cSTA_TURNBusy: INT := 215;
	cSTA_TURN: INT := RAX_CmdState.cCMD_TURN;
END_VAR

// POUs/Controller/Lvl1/BCH (Barcode with DataChannel)/BCH_CmdState
VAR_GLOBAL CONSTANT
	cCMD_READ: INT := 200;
	cSUB_WAITPAPER: INT := 300;
	cSUB_BARCODEREADstart: INT := 310;
	cSUB_BARCODREREADbusy: INT := 311;
	cSUB_BARCODREREAD: INT := 312;
	cSUB_WAITPAPERGONE: INT := 313;
	cSUB_WAITPAPERGONEDELAY: INT := 314;
END_VAR

// POUs/Controller/Lvl1/MDC [Malteser Drive Controller]/MDC_CmdState
VAR_GLOBAL CONSTANT
	///ctrl commands definitions
	///specific commands >200 - every command has to be a even number
	cCMD_INITIALIZE			: INT := 202;
	cCMD_TURN    			: INT := 204;
	cCMD_PREPOSITION		: INT := 210;
	
	///ctrl specific states definitions
	cSTA_InitializeBusy		: INT := 201;
	cSTA_InPositionBusy		: INT := 203;
	cSTA_InPosition			: INT := 205;
	cSTA_StartTurnBusy		: INT := 207;
	cSTA_TurnBusy			: INT := 209;
	cSTA_PREPOSITIONbusy	: INT := 220;
	cSTA_PREPOSITION		: INT := 221;
	cSTA_TURNDONE			: INT := 222;
	
	cSUB_TURNbusy			: INT := 300;
	cSUB_STOPbusy			: INT := 301;
	cSUB_FINDHOLEbusy		: INT := 302;
END_VAR

// POUs/Controller/Lvl1/OVN (Oven)/OVN_CmdState
VAR_GLOBAL CONSTANT
	///ctrl commands definitions
	///specific commands >200 - every command has to be a even number
	cCMD_BELTONLY: INT := 202;
	///ctrl specific states definitions
	cSTA_BELTONLYBusy: INT := 201;
	cSTA_BELTONLY: INT := 202;
	cSUB_WAITOFF: INT := 300;
	cSUB_WAITPAPER: INT := 301;
	cSUB_DONE: INT := 302;
END_VAR

// POUs/Controller/Lvl1/PTB [Paper Transport Belt]/PTB_CmdState
VAR_GLOBAL CONSTANT
	///ctrl commands definitions
	cCMD_EJECTPAPER			: INT := 202;
	cCMD_STACKPAPER			: INT := 204;
	///specific commands >200 - every command has to be a even number
	///ctrl specific states definitions
	cSTA_EJECTPAPERbusy		: INT := 201;
	cSTA_EJECTPAPER			: INT := 202;
	cSTA_STACKPAPERbusy		: INT := 203;
	cSTA_STACKPAPER			: INT := 204;

	///ctrl specific sub states definitions
	cSUB_EMPTYstart					: INT := 300;
	cSUB_EMPTYWAITPAPERbusy			: INT := 301;
	cSUB_EMPTYWAITPAPERdebounce		: INT := 302;
	cSUB_EMPTYWAITPAPERGONEbusy		: INT := 303;
	cSUB_EMPTYWAITPAPERGONEdebounce	: INT := 304;
	cSUB_EMPTYWAITDRIVESTOPED		: INT := 305;
	cSUB_WAITPAPER  				: INT := 306;
	cSUB_WAITPAPERGONE  			: INT := 307;
	cSUB_STARTSTACKDELAY			: INT := 308;
	cSUB_PAPERDISTANCEstart			: INT := 309;
	cSUB_PAPERDISTANCEbusy			: INT := 310;
	cSUB_PAPERDISTANCESTOPbusy		: INT := 311;
	cSUB_STARTENTRYDRIVEbusy		: INT := 312;
	cSUB_STARTENTRYDRIVE			: INT := 313;
END_VAR

// POUs/Controller/Lvl2/PBC [Paper Buffer Controller]/PBC_CmdState
VAR_GLOBAL CONSTANT
	///ctrl specific command definitions
	cCMD_SINGLE			: INT := 202;
	cCMD_MANUALSTART	: INT := 204;
	///ctrl specific states definitions
	cSTA_INITbusy		: INT := 205;
	cSUB_WAITPAPER: INT := 300;
	cSUB_POSITIONbusy: INT := 301;
	cSUB_POSITIONSTOPbusy: INT := 302;
	cSUB_EVALUATEEJECT: INT := 303;
	cSUB_EJECTbusy: INT := 304;
	cSUB_EJECTSTOPbusy: INT := 305;
	cSUB_POSITIONSTARTbusy: INT := 306;
	cSUB_EJECTSTARTbusy: INT := 307;
	cSUB_READYEJECT: INT := 308;
	cSUB_WAITPAPERGONETABLE: INT := 309;
	///	cSUB_BARCODEREADstart	: INT := 310;
	///	cSUB_BARCODREREADbusy	: INT := 311;
	///	cSUB_BARCODREREAD  		: INT := 312;
	cSUB_POSITIONRETRYDELAY: INT := 313;
	cSUB_POSITIONRETRYSTOP: INT := 314;
END_VAR

// POUs/Controller/Lvl2/PCE [Paper Belt Corner Element]/PCE_CmdState
VAR_GLOBAL CONSTANT
	///ctrl commands definitions
	///specific commands >200 - every command has to be a even number
	///ctrl specific states definitions
	cSUB_PAPERENTRY: INT := 300;
	cSUB_PAPERENTRYDelay: INT := 301;
	cSUB_PAPEREXIT: INT := 302;
END_VAR

// POUs/Controller/Lvl2/PST [Paper Stacker]/PST_CmdState
VAR_GLOBAL CONSTANT
	/// specific commands >200 - every command has to be a even number
	/// ctrl commands definitions
	cCMD_EJECT: INT := 202;
	/// main states
	cSTA_EJECTbusy: INT := 201;
	/// sub states
	cSUB_WAITNEWPAPERDETECTED: INT := 300;
	cSUB_DELAYREADBARCODEBusy: INT := 301;
	cSUB_RETRYREADBARCODE: INT := 302;
	cSUB_READBARCODEbusy: INT := 303;
	cSUB_CHECKEJECTCONDITIONS: INT := 304;
	cSUB_DELAYSTACKEJECTBusy: INT := 305;
	cSUB_MOVEBELTEJECTDIRECTIONBusy: INT := 306;
	cSUB_STOPBELTBusy: INT := 307;
	cSUB_WAITBEFOREMOVINGREVERSE: INT := 308;
	cSUB_MOVEBELTREVERSEBusy: INT := 309;
	cSUB_DONE: INT := 999;
END_VAR

// POUs/Controller/Lvl2/PTS [Paper Turning Station]/PTS_CmdState
VAR_GLOBAL CONSTANT
	///ctrl specific command definitions
	cCMD_TURN: INT := 202;
	cCMD_STANDBY: INT := 204;
	///ctrl specific states definitions
	cSTA_STANDBYBusy: INT := 203;
	cSTA_STANDBY: INT := 204;
	cSTA_PaperDelayBusy: INT := 205;
	cSTA_TurnPaperBusy: INT := 207;
	cSTA_WaitPaperGone: INT := 209;
	cSTA_EmptyDelayBusy: INT := 211;
	cSTA_TurnEmptyBusy: INT := 213;
	cSTA_InitializeBusy: INT := 215;
	cSTA_WaitPaper: INT := 217;
	cSTA_GetItemBusy: INT := 219;
	/// ctrl specific substates definitions
	cSUB_WAIT_START: INT := 300;
	cSUB_WAIT_DONE: INT := 301;
	cSUB_TURNbusy: INT := 302;
	cSUB_TURNDONE: INT := 303;
	cSUB_PREPOSITIONbusy: INT := 304;
	cSUB_DELAYbusy: INT := 305;
	cSUB_WAITPAPERGONEbusy: INT := 306;
	/// Other Constants
	cPTS_MAX_AUTOPOS: UINT := 5;
	cPTS_MAX_DISTRIBUTION: INT := 2;
END_VAR

// POUs/Controller/Lvl2/PTS [Paper Turning Station]/PTS_Persistent
VAR_GLOBAL PERSISTENT
	udiPTS_Counter_Persistent: UDINT;	// Count of turn movements. This is a persistent variable, reset only with reset origin
END_VAR

// POUs/Controller/Utility/Data Channel/OvenMessage/OvenConst
VAR_GLOBAL CONSTANT
	cRECVDATACHANNELBUFFER: INT := 20;
END_VAR

// POUs/Controller/Utility/LookupTable/LUT_Constants
VAR_GLOBAL CONSTANT
	/// max size of lookup table
	MaxLookupSize: INT := 20;
END_VAR

// Version/Global_Version
// This function has been automatically generated from the project information.
VAR_GLOBAL CONSTANT
	{attribute 'const_non_replaced'}
	stLibVersion_BasePpt : ST_LibVersion := (iMajor := 0, iMinor := 0, iBuild := 0, iRevision := 76, sVersion := '0.0.0.76');
END_VAR

// POUs/Controller/Driver/IBH (IBH Link)/FB_IBH
FUNCTION_BLOCK FB_IBH EXTENDS FB_CtrlBase
VAR_OUTPUT
	/// Status 
	Out_iStatus: INT;
	/// Machine off 
	Out_bOff: BOOL;
	/// Band on 
	Out_bBeltOn: BOOL;
	/// Manual Mode 
	Out_bManual: BOOL;
	/// Standart drying process 
	Out_bRun: BOOL;
	/// Set Parameter 
	Out_bSetParam: BOOL;
	/// Get Parameter 
	Out_bGetParam: BOOL;
	/// Resetting error 
	Out_bAckError: BOOL;
	/// Actual temperature in deci °C 
	Out_adiTemp_dc: ARRAY[0..(MAX_NUMBER_OF_OVEN_MODULES - 1)] OF DINT;
	/// Aactual airflow in % 
	Out_adiAir_p: ARRAY[0..(MAX_NUMBER_OF_OVEN_MODULES - 1)] OF DINT;
	/// Actual belt speed in mm/min 
	Out_diSpeed_mm_min: DINT;
	/// 1=Information, 2=Warning, 3=Error 
	Out_iErrorLevel: INT;
	/// Error ID (e.g. 100=temperature overflow) 
	Out_iErrorID: INT;
	Out_bDriverConnected: BOOL;
	Out_bDriverError: BOOL;
	Out_udiDriverErrorID: UDINT;
END_VAR
VAR
	/// Specific interface struct for public access
	SIf: T_Ctrl_SIf_IBH;
	/// Turns oven off 
	iOff: INT;
	/// Turns belt on 
	iBeltOn: INT;
	/// Puts oven to manual  
	iManual: INT;
	/// Standart drying process 
	iRun: INT;
	/// Set Parameter 
	iSetParam: INT;
	/// Get Parameter 
	iGetParam: INT;
	/// Temperature in deci °C 
	adiTemp_dc: ARRAY[0..(MAX_NUMBER_OF_OVEN_MODULES - 1)] OF DINT;
	/// Airflow in % 
	adiAir_p: ARRAY[0..(MAX_NUMBER_OF_OVEN_MODULES - 1)] OF DINT;
	/// Belt speed in mm/min 
	diSpeed_mm_min: DINT;
	/// Try to reset error 
	iAckError: INT;
	bIncrementSetParam: BOOL;
	bRememberIncrementSetParam: BOOL;
	fbOpen: Tc2_S5S7Com.FB_NLinkOpen;
	fbWrite: Tc2_S5S7Com.FB_NLinkWrite;
	fbFetch: Tc2_S5S7Com.FB_NLinkFetch;
	fbClose: Tc2_S5S7Com.FB_NLinkClose;
	/// Communication link handle 
	hLink: T_HNLINK;
	/// read data buffer 
	anReadBuffer: ARRAY[0..(READ_BUFFER_LENGTH - 1)] OF BYTE;
	/// data to write 
	anWriteBuffer: ARRAY[0..(WRITE_BUFFER_LENGTH - 1)] OF BYTE;
	
	// simulation
	iSimStatus: INT;
	bSimOff: BOOL;
	bSimBeltOn: BOOL;
	bSimManual: BOOL;
	bSimRun: BOOL;
END_VAR

(*__________________________________________________________________________________________________
¦	
¦	Vistaprint Schweiz GmbH
¦	CH - 8401 Winterthur
¦
¦	www.vistaprint.ch - info@vistaprint.ch
¦___________________________________________________________________________________________________

Function desription:
IBH Link Connection Implementation

History:
Version		Date			Author		Comment
---------------------------------------------------------------------------------------------------
0.00.1		09.01.2014		BB			Start history
___________________________________________________________________________________________________*)

SUPER^();

{attribute 'object_name' := 'Always'}
METHOD PROTECTED Always : BOOL
VAR
	fbOVN: INT;
END_VAR
// ----------------------------------------------------------------------------------
// Conditions Always
IF (me.bolChangeBackToAUTO=TRUE) THEN // switch mode to automatic switch off controller
	me.StateMachine.intStateNext := cSTA_OFFBusy;
	me.bolChangeBackToAUTO := FALSE;
END_IF

IF (CIf.SwCfg.bolExist=FALSE) THEN // hardware of controller does not exist
	me.StateMachine.intStateNext := cSTA_SINGLE_ANSWER;
ELSE
	IF (((me.StateMachine.intState=cSTA_INITIALIZED) OR (me.intCmd=cCMD_PON)) 
		AND (me.StateMachine.intState<>cSTA_PONBusy) AND (me.StateMachine.intState<>cSTA_PON)
		AND (me.StateMachine.intState<>cSTA_ERROR) AND (me.StateMachine.intState<>cSTA_ERRORQuit) 
		AND (me.StateMachine.intState<>cSTA_EOFF) AND (me.StateMachine.intState<>cSTA_EOFFBusy)) THEN // switch after startup to PONBusy
		me.StateMachine.intStateNext := cSTA_PONBusy;
		
	ELSIF (((me.Alarm.eActivAlmClass=E_AlmClass.EOFF) OR (me.intCmd=cCMD_EOFF)) 
		AND (me.StateMachine.intState<>cSTA_ERROR) AND (me.StateMachine.intState<>cSTA_ERRORQuit) 
		AND (me.StateMachine.intState<>cSTA_EOFF) AND (me.StateMachine.intState<>cSTA_EOFFBusy)
		AND (me.StateMachine.intState>cSTA_PON)) THEN
		me.StateMachine.intStateNext := cSTA_EOFFBusy;
	
	ELSIF (((me.Alarm.eActivAlmClass=E_AlmClass.OFF) (*OR (me.intCmd=cCMD_OFF)*))
		AND (me.StateMachine.intState<>cSTA_ERROR) AND (me.StateMachine.intState<>cSTA_ERRORQuit)
		AND (me.StateMachine.intState<>cSTA_EOFF) AND (me.StateMachine.intState<>cSTA_EOFFBusy)
		AND (me.StateMachine.intState<>cSTA_OFF) AND (me.StateMachine.intState<>cSTA_OFFBusy)
		AND (me.StateMachine.intState>cSTA_PON)) THEN
		me.StateMachine.intStateNext := cSTA_OFFBusy;
	
	END_IF
	
	IF		NOT CIf.SwCfg.bolEnable
		AND (me.StateMachine.intState<>cSTA_OFF)
		AND (me.StateMachine.intState<>cSTA_OFFBusy) THEN
		CIf.Job.intACmd := cCMD_OFF;
	END_IF
	
	Out_bDriverConnected := FALSE;
	IF		(me.StateMachine.intState=cSTA_WRITE) OR (me.StateMachine.intState=cSTA_WRITEBusy)
		OR	(me.StateMachine.intState=cSTA_READ) OR (me.StateMachine.intState=cSTA_READBusy) THEN
		Out_bDriverConnected := TRUE;
	END_IF
	
END_IF

// ----------------------------------------------------------------------------------
// overrule error always from base -> no EOFF State!! in EOFF go to OFF
IF (me.StateMachine.intStateNext = cSTA_EOFFBusy) THEN
	IF (me.StateMachine.intState = cSTA_OFF) THEN
		me.StateMachine.intStateNext := cSTA_OFF;
	ELSE // stay in OFF
		me.StateMachine.intStateNext := cSTA_OFFBusy;
	END_IF
END_IF
END_METHOD

